// POUs/BACnet Objects/Local (Server)/ADS/FB_BACnet_BinaryOutput_ADS
FUNCTION_BLOCK FB_BACnet_BinaryOutput_ADS
VAR_INPUT
	bEnablePV			: BOOL; (* enable PV write commands *)
	bNullPV				: BOOL; (* clear priority entry *)
	bPV					: BOOL; (* present value bool type *)
	bManual				: BOOL; (* FALSE --> TRUE: write present_value immediately, FALSE: only write present_value on-change, TRUE: write present_value on-change and when device turns operational *)
	ePriority			: E_BACNETPRIORITY := BACNETPRIORITY_12;
END_VAR
VAR_IN_OUT
	Device				: FB_BACnet_Device;
END_VAR
VAR_OUTPUT
	bReady				: BOOL;
	bPvDone				: BOOL; (* present_value written over ADS *)
	bPresentValue		: BOOL;
	bOverridden			: BOOL;
	bOutOfService		: BOOL;
	bFault				: BOOL;
	bInAlarm			: BOOL;
	tObjectID			: T_BACnet_ObjectIdentifier := 16#FFFFFFFF;
	bError				: BOOL;
	nErrorId			: UINT;
	nAdsErrorId			: UDINT;
END_VAR
VAR
	_ObjectId AT%I*: DWORD;				(* ~(BACnet_ObjectIdentifier	:		: LINK) *)
	_PresentValue AT%I*: WORD; 			(* ~(BACnet_PresentValue 		:		: )
								   			(BACnet_ObjectType 			: BO	: )	*)
    _PresentValue_Ads : WORD;
	_StatusFlags AT%I*: WORD; 			(* ~(BACnet_StatusFlags 		:		: )	*)
	_StatusFlagsBits : ST_BACnet_StatusFlags;
	_nUpdateCount : UDINT := 0;
	_WriteProp : FB_BACnet_WriteProp;
	_rtrigManual : R_TRIG;
	_bNullPvOld : BOOL;
	_nObjType : E_BACNETOBJECTTYPE;
END_VAR

(* update server device *)
IF (Device._nUpdateCount = _nUpdateCount) THEN
	Device();
END_IF
(* remind current number of update counter *)
_nUpdateCount := Device._nUpdateCount;

(* trigger on manual flag *)
_rtrigManual(CLK:= bManual, Q=> );

(* decode object type *)
_nObjType := F_BACnet_GetObjType(_ObjectId);

IF Device.bFirstCycle THEN
	(* first call of the server device since reboot/reset *)
	bReady := FALSE;
	bPvDone := FALSE;

ELSIF _nObjType <> BACnetObjectType_BinaryOutput THEN
	(* wrong mapped object type *)
	nErrorId := BACnet_ERR_INVALID_OBJECTTYPE;
	bReady := FALSE;
	bPvDone := FALSE;

ELSIF (_StatusFlags < 4) THEN
	(* wrong mapping *)
	nErrorId := BACnet_ERR_WRONG_MAPPING;
	bReady := FALSE;
	bPvDone := FALSE;

ELSIF Device.bOperational THEN

	IF Device.stAdsConn.bValid THEN
		(* write present_value on manual trigger, on-change and on operational recover *)
		IF	(		bEnablePV
				AND	(		(bPV <> F_BinPV_To_Bool(TO_INT(_PresentValue_Ads)))
						OR	((NOT bReady) AND bManual)
						OR	(bNullPV <> _bNullPvOld)
						OR	_rtrigManual.Q
					)
			)
		THEN
			_WriteProp.bExecute := TRUE;
			bPvDone := FALSE;
			(* write depending on enable state *)
			_PresentValue_Ads := TO_WORD(F_Bool_To_BinPV(TRUE, bNullPV, bPV));
			_bNullPvOld := bNullPV;
		END_IF

		(* ready state *)
		IF (nAdsErrorId = 0) THEN
			bReady := TRUE;
			nErrorId := BACnet_ERR_NO_ERROR;
		END_IF

	ELSE
		(* invalid ADS connection *)
		bReady := FALSE;
		nErrorId := BACnet_ERR_INVALID_ADS_CONN;
		bPvDone := FALSE;
	END_IF


	(* present value *)
	bPresentValue := F_BinPV_To_Bool(TO_INT(_PresentValue));

	(* build bit states *)
	_StatusFlagsBits := F_BACnet_StatusFlags(_StatusFlags);

	(* copy states to output *)
	bOverridden := _StatusFlagsBits.overridden;
	bOutOfService := _StatusFlagsBits.out_of_service;
	bFault := _StatusFlagsBits.fault;
	bInAlarm := _StatusFlagsBits.in_alarm;
	tObjectID := _ObjectId;

ELSE
	(* server device not ready, reset local ready also *)
	bReady := FALSE;
	nErrorId := BACnet_ERR_OPERATIONAL;
	bPvDone := FALSE;
END_IF

(* call write property command *)
_WriteProp(
	BACnetDevicePort	:= Device.stAdsConn.nAmsPort,
	bExecute			:= ,
	sNetId				:= Device.stAdsConn.sAmsNetId,
	ObjectType			:= _nObjType,
	PropertyID			:= BACnetPropertyIdentifier_PresentValue,
	Priority			:= ePriority,
	DataType			:= BACnetDataType_BinaryPV,
	ObjectInstance		:= F_BACnet_GetObjInstance(_ObjectId),
	ptrValue			:= ADR(_PresentValue_Ads),
	nLenValue			:= SIZEOF(_PresentValue_Ads),
	bDone				=> ,
	bBusy				=> ,
	bError				=> ,
	nErrID				=> );

(* set done flag *)
IF _WriteProp.bExecute AND (NOT _WriteProp.bBusy) THEN
	(* check if command was finished with error *)
	IF _WriteProp.bError THEN
		bPvDone		:= FALSE;
		bReady		:= FALSE;
		nErrorId	:= BACnet_ERR_ADS_Write;
	ELSE
		(* successful written *)
		bPvDone		:= TRUE;
	END_IF
	nAdsErrorId := _WriteProp.nErrID;
	(* reset execution bit *)
	_WriteProp(bExecute := FALSE);
END_IF

(* set error flag *)
bError := (nErrorId <> BACnet_ERR_NO_ERROR) OR (nAdsErrorId <> 0);

END_FUNCTION_BLOCK

// POUs/BACnet Objects/Local (Server)/ADS/FB_BACnet_BinaryValue_ADS
FUNCTION_BLOCK FB_BACnet_BinaryValue_ADS
VAR_INPUT
	bEnablePV			: BOOL; (* enable PV write commands *)
	bNullPV				: BOOL; (* clear priority entry *)
	bPV					: BOOL; (* present value bool type *)
	bManual				: BOOL; (* FALSE --> TRUE: write present_value immediately, FALSE: only write present_value on-change, TRUE: write present_value on-change and when device turns operational *)
	ePriority			: E_BACNETPRIORITY := BACNETPRIORITY_12;
END_VAR
VAR_IN_OUT
	Device				: FB_BACnet_Device;
END_VAR
VAR_OUTPUT
	bReady				: BOOL;
	bPvDone				: BOOL; (* present_value written over ADS *)
	bPresentValue		: BOOL;
	bOverridden			: BOOL;
	bOutOfService		: BOOL;
	bFault				: BOOL;
	bInAlarm			: BOOL;
	tObjectID			: T_BACnet_ObjectIdentifier := 16#FFFFFFFF;
	bError				: BOOL;
	nErrorId			: UINT;
	nAdsErrorId			: UDINT;
END_VAR
VAR
	_ObjectId AT%I*: DWORD;				(* ~(BACnet_ObjectIdentifier		:		: LINK) *)
	_PresentValue AT%I*: WORD; 			(* ~(BACnet_PresentValue 			:		: )
								   			(BACnet_ObjectType 				: BV	: )	*)
    _PresentValue_Ads : WORD;
	_StatusFlags AT%I*: WORD; 			(* ~(BACnet_StatusFlags 			:		: )	*)
	_StatusFlagsBits : ST_BACnet_StatusFlags;
	_nUpdateCount : UDINT := 0;
	_WriteProp : FB_BACnet_WriteProp;
	_rtrigManual : R_TRIG;
	_bNullPvOld : BOOL;
	_nObjType : E_BACNETOBJECTTYPE;
END_VAR

(* update server device *)
IF (Device._nUpdateCount = _nUpdateCount) THEN
	Device();
END_IF
(* remind current number of update counter *)
_nUpdateCount := Device._nUpdateCount;

(* trigger on manual flag *)
_rtrigManual(CLK:= bManual, Q=> );

(* decode object type *)
_nObjType := F_BACnet_GetObjType(_ObjectId);

IF Device.bFirstCycle THEN
	(* first call of the server device since reboot/reset *)
	bReady := FALSE;
	bPvDone := FALSE;

ELSIF _nObjType <> BACnetObjectType_BinaryValue THEN
	(* wrong mapped object type *)
	nErrorId := BACnet_ERR_INVALID_OBJECTTYPE;
	bReady := FALSE;
	bPvDone := FALSE;

ELSIF (_StatusFlags < 4) THEN
	(* wrong mapping *)
	nErrorId := BACnet_ERR_WRONG_MAPPING;
	bReady := FALSE;
	bPvDone := FALSE;

ELSIF Device.bOperational THEN

	IF Device.stAdsConn.bValid THEN
		(* write present_value on manual trigger, on-change and on operational recover *)
		IF (		bEnablePV
				AND	(		(bPV <> F_BinPV_To_Bool(TO_INT(_PresentValue_Ads)))
						OR	((NOT bReady) AND bManual)
						OR	(bNullPV <> _bNullPvOld)
						OR	_rtrigManual.Q
					)
			)
		THEN
			_WriteProp.bExecute := TRUE;
			bPvDone := FALSE;
			(* write depending on enable state *)
			_PresentValue_Ads := to_word(F_Bool_To_BinPV(TRUE, bNullPV, bPV));
			_bNullPvOld := bNullPV;
		END_IF

		(* ready state *)
		IF (nAdsErrorId = 0) THEN
			bReady := TRUE;
			nErrorId := BACnet_ERR_NO_ERROR;
		END_IF

	ELSE
		(* invalid ADS connection *)
		bReady := FALSE;
		nErrorId := BACnet_ERR_INVALID_ADS_CONN;
		bPvDone := FALSE;
	END_IF

	(* present value *)
	bPresentValue := F_BinPV_To_Bool(TO_INT(_PresentValue));

	(* build bit states *)
	_StatusFlagsBits := F_BACnet_StatusFlags(_StatusFlags);

	(* copy states to output *)
	bOverridden := _StatusFlagsBits.overridden;
	bOutOfService := _StatusFlagsBits.out_of_service;
	bFault := _StatusFlagsBits.fault;
	bInAlarm := _StatusFlagsBits.in_alarm;
	tObjectID := _ObjectId;

ELSE
	(* server device not ready, reset local ready also *)
	bReady := FALSE;
	nErrorId := BACnet_ERR_OPERATIONAL;
	bPvDone := FALSE;
END_IF

(* call write property command *)
_WriteProp(
	BACnetDevicePort	:= Device.stAdsConn.nAmsPort,
	bExecute			:= ,
	sNetId				:= Device.stAdsConn.sAmsNetId,
	ObjectType			:= _nObjType,
	PropertyID			:= BACnetPropertyIdentifier_PresentValue,
	Priority			:= ePriority,
	DataType			:= BACnetDataType_BinaryPV,
	ObjectInstance		:= F_BACnet_GetObjInstance(_ObjectId),
	ptrValue			:= ADR(_PresentValue_Ads),
	nLenValue			:= SIZEOF(_PresentValue_Ads),
	bDone				=> ,
	bBusy				=> ,
	bError				=> ,
	nErrID				=> );

(* set done flag *)
IF _WriteProp.bExecute AND (NOT _WriteProp.bBusy) THEN
	(* check if command was finished with error *)
	IF _WriteProp.bError THEN
		bPvDone		:= FALSE;
		bReady		:= FALSE;
		nErrorId	:= BACnet_ERR_ADS_Write;
	ELSE
		(* successful written *)
		bPvDone		:= TRUE;
	END_IF
	nAdsErrorId := _WriteProp.nErrID;
	(* reset execution bit *)
	_WriteProp(bExecute := FALSE);
END_IF

(* set error flag *)
bError := (nErrorId <> BACnet_ERR_NO_ERROR) OR (nAdsErrorId <> 0);

END_FUNCTION_BLOCK

// POUs/BACnet Objects/Local (Server)/ADS/FB_BACnet_MultiStateOutput_ADS
FUNCTION_BLOCK FB_BACnet_MultiStateOutput_ADS
VAR_INPUT
	bEnablePV			: BOOL; (* enable PV write commands *)
	bNullPV				: BOOL; (* clear priority entry *)
	nPV					: UDINT; (* number for priority x, when input bEnablePV is TRUE and bNullPV is FALSE *)
	bManual				: BOOL; (* FALSE --> TRUE: write present_value immediately, FALSE: only write present_value on-change, TRUE: write present_value on-change and when device turns operational *)
	ePriority			: E_BACNETPRIORITY := BACNETPRIORITY_12;
END_VAR
VAR_IN_OUT
	Device				: FB_BACnet_Device;
END_VAR
VAR_OUTPUT
	bReady				: BOOL;
	bPvDone				: BOOL; (* present_value written over ADS *)
	nPresentValue		: UDINT;
	bOverridden			: BOOL;
	bOutOfService		: BOOL;
	bFault				: BOOL;
	bInAlarm			: BOOL;
	nNbrOfStates		: UDINT;
	tObjectID			: T_BACnet_ObjectIdentifier := 16#FFFFFFFF;
	bError				: BOOL;
	nErrorId			: UINT;
	nAdsErrorId			: UDINT;
END_VAR
VAR
	_StatusFlags AT%I*: WORD; 				(* ~(BACnet_StatusFlags			:		: )	*)
	_PresentValue AT%I*: UDINT; 			(* ~(BACnet_PresentValue 		:		: )
								   				(BACnet_ObjectType			: MO	: )	*)
	_NumberOfStates AT%I*: UDINT;			(* ~(BACnet_NumberOfStates		:		: )	*)
	_ObjectId AT%I*: DWORD;					(* ~(BACnet_ObjectIdentifier	:		: LINK) *)
	_StatusFlagsBits : ST_BACnet_StatusFlags;
    _PresentValue_Ads : UDINT;
	_nUpdateCount : UDINT := 0;
	_WriteProp : FB_BACnet_WriteProp;
	_rtrigManual : R_TRIG;
	_bNullPvOld : BOOL;
	_nObjType : E_BACNETOBJECTTYPE;
END_VAR

(* update server device *)
IF (Device._nUpdateCount = _nUpdateCount) THEN
	Device();
END_IF
(* remind current number of update counter *)
_nUpdateCount := Device._nUpdateCount;

(* trigger on manual flag *)
_rtrigManual(CLK:= bManual, Q=> );

(* decode object type *)
_nObjType := F_BACnet_GetObjType(_ObjectId);

IF Device.bFirstCycle THEN
	(* first call of the server device since reboot/reset *)
	bReady := FALSE;
	bPvDone := FALSE;

ELSIF _nObjType <> BACnetObjectType_MultiStateOutput THEN
	(* wrong mapped object type *)
	nErrorId := BACnet_ERR_INVALID_OBJECTTYPE;
	bReady := FALSE;
	bPvDone := FALSE;

ELSIF (_StatusFlags < 4) THEN
	(* wrong mapping *)
	nErrorId := BACnet_ERR_WRONG_MAPPING;
	bReady := FALSE;
	bPvDone := FALSE;

ELSIF Device.bOperational THEN

	IF Device.stAdsConn.bValid THEN
		(* write present_value on manual trigger, on-change and on operational recover *)
		IF		bEnablePV
			AND	(		_rtrigManual.Q
					OR	(nPV <> _PresentValue_Ads)
					OR	((NOT bReady) AND bManual)
					OR	(bNullPV <> _bNullPvOld)
				)
		THEN
			_WriteProp.bExecute := TRUE;
			bPvDone := FALSE;
			(* write depending on enable state *)
			IF bNullPV THEN
				_PresentValue_Ads := 0;
			ELSE
				_PresentValue_Ads := nPV;
			END_IF
			_bNullPvOld := bNullPV;
		END_IF

		(* ready state *)
		IF (nAdsErrorId = 0) THEN
			bReady := TRUE;
			nErrorId := BACnet_ERR_NO_ERROR;
		END_IF

	ELSE
		(* invalid ADS connection *)
		bReady := FALSE;
		nErrorId := BACnet_ERR_INVALID_ADS_CONN;
		bPvDone := FALSE;
	END_IF

	(* present value *)
	nPresentValue := _PresentValue;

	(* build bit states *)
	_StatusFlagsBits := F_BACnet_StatusFlags(_StatusFlags);

	(* copy states to output *)
	bOverridden := _StatusFlagsBits.overridden;
	bOutOfService := _StatusFlagsBits.out_of_service;
	bFault := _StatusFlagsBits.fault;
	bInAlarm := _StatusFlagsBits.in_alarm;
	tObjectID := _ObjectId;

	(* number of states *)
	nNbrOfStates := _NumberOfStates;

ELSE
	(* server device not ready, reset local ready also *)
	bReady := FALSE;
	nErrorId := BACnet_ERR_OPERATIONAL;
	bPvDone := FALSE;
END_IF

(* call write property command *)
_WriteProp(
	BACnetDevicePort	:= Device.stAdsConn.nAmsPort,
	bExecute			:= ,
	sNetId				:= Device.stAdsConn.sAmsNetId,
	ObjectType			:= _nObjType,
	PropertyID			:= BACnetPropertyIdentifier_PresentValue,
	Priority			:= ePriority,
	DataType			:= BACnetDataType_UnsignedInteger,
	ObjectInstance		:= F_BACnet_GetObjInstance(_ObjectId),
	ptrValue			:= ADR(_PresentValue_Ads),
	nLenValue			:= SIZEOF(_PresentValue_Ads),
	bDone				=> ,
	bBusy				=> ,
	bError				=> ,
	nErrID				=> );

(* set done flag *)
IF _WriteProp.bExecute AND (NOT _WriteProp.bBusy) THEN
	(* check if command was finished with error *)
	IF _WriteProp.bError THEN
		bPvDone		:= FALSE;
		bReady		:= FALSE;
		nErrorId	:= BACnet_ERR_ADS_Write;
	ELSE
		(* successful written *)
		bPvDone		:= TRUE;
	END_IF
	nAdsErrorId := _WriteProp.nErrID;
	(* reset execution bit *)
	_WriteProp(bExecute := FALSE);
END_IF

(* set error flag *)
bError := (nErrorId <> BACnet_ERR_NO_ERROR) OR (nAdsErrorId <> 0);

END_FUNCTION_BLOCK

// POUs/BACnet Objects/Local (Server)/ADS/FB_BACnet_MultiStateValue_ADS
FUNCTION_BLOCK FB_BACnet_MultiStateValue_ADS
VAR_INPUT
	bEnablePV			: BOOL; (* enable PV write commands *)
	bNullPV				: BOOL; (* clear priority entry *)
	nPV					: UDINT; (* number for priority x, when input bEnablePV is TRUE and bNullPV is FALSE *)
	bManual				: BOOL; (* FALSE --> TRUE: write present_value immediately, FALSE: only write present_value on-change, TRUE: write present_value on-change and when device turns operational *)
	ePriority			: E_BACNETPRIORITY := BACNETPRIORITY_12;
END_VAR
VAR_IN_OUT
	Device				: FB_BACnet_Device;
END_VAR
VAR_OUTPUT
	bReady				: BOOL;
	bPvDone				: BOOL; (* present_value written over ADS *)
	nPresentValue		: UDINT;
	bOverridden			: BOOL;
	bOutOfService		: BOOL;
	bFault				: BOOL;
	bInAlarm			: BOOL;
	nNbrOfStates		: UDINT;
	tObjectID			: T_BACnet_ObjectIdentifier := 16#FFFFFFFF;
	bError				: BOOL;
	nErrorId			: UINT;
	nAdsErrorId			: UDINT;
END_VAR
VAR
	_StatusFlags AT%I*: WORD; 				(* ~(BACnet_StatusFlags 	:		: )	*)
	_PresentValue AT%I*: UDINT; 			(* ~(BACnet_PresentValue 	:		: )
								   				(BACnet_ObjectType 		: MV	: )	*)
	_NumberOfStates AT%I*: UDINT;			(* ~(BACnet_NumberOfStates	:		: )	*)
	_ObjectId AT%I*: DWORD;					(* ~(BACnet_ObjectIdentifier:		: LINK) *)
	_StatusFlagsBits : ST_BACnet_StatusFlags;
    _PresentValue_Ads : UDINT;
	_nUpdateCount : UDINT := 0;
	_WriteProp : FB_BACnet_WriteProp;
	_rtrigManual : R_TRIG;
	_bNullPvOld : BOOL;
	_nObjType : E_BACNETOBJECTTYPE;
END_VAR

(* update server device *)
IF (Device._nUpdateCount = _nUpdateCount) THEN
	Device();
END_IF
(* remind current number of update counter *)
_nUpdateCount := Device._nUpdateCount;

(* trigger on manual flag *)
_rtrigManual(CLK:= bManual, Q=> );

(* decode object type *)
_nObjType := F_BACnet_GetObjType(_ObjectId);

IF Device.bFirstCycle THEN
	(* first call of the server device since reboot/reset *)
	bReady := FALSE;
	bPvDone := FALSE;

ELSIF _nObjType <> BACnetObjectType_MultiStateValue THEN
	(* wrong mapped object type *)
	nErrorId := BACnet_ERR_INVALID_OBJECTTYPE;
	bReady := FALSE;
	bPvDone := FALSE;

ELSIF (_StatusFlags < 4) THEN
	(* wrong mapping *)
	nErrorId := BACnet_ERR_WRONG_MAPPING;
	bReady := FALSE;
	bPvDone := FALSE;

ELSIF Device.bOperational THEN

	IF Device.stAdsConn.bValid THEN
		(* write present_value on manual trigger, on-change and on operational recover *)
		IF		bEnablePV
			AND	(		_rtrigManual.Q
					OR	(nPV <> _PresentValue_Ads)
					OR	((NOT bReady) AND bManual)
					OR	(bNullPV <> _bNullPvOld)
				)
		THEN
			_WriteProp.bExecute := TRUE;
			bPvDone := FALSE;
			(* write depending on enable state *)
			IF bNullPV THEN
				_PresentValue_Ads := 0;
			ELSE
				_PresentValue_Ads := nPV;
			END_IF
			_bNullPvOld := bNullPV;
		END_IF

		(* ready state *)
		IF (nAdsErrorId = 0) THEN
			bReady := TRUE;
			nErrorId := BACnet_ERR_NO_ERROR;
		END_IF

	ELSE
		(* invalid ADS connection *)
		bReady := FALSE;
		nErrorId := BACnet_ERR_INVALID_ADS_CONN;
		bPvDone := FALSE;
	END_IF

	(* present value *)
	nPresentValue := _PresentValue;

	(* build bit states *)
	_StatusFlagsBits := F_BACnet_StatusFlags(_StatusFlags);

	(* copy states to output *)
	bOverridden := _StatusFlagsBits.overridden;
	bOutOfService := _StatusFlagsBits.out_of_service;
	bFault := _StatusFlagsBits.fault;
	bInAlarm := _StatusFlagsBits.in_alarm;
	tObjectID := _ObjectId;

	(* number of states *)
	nNbrOfStates := _NumberOfStates;

ELSE
	(* server device not ready, reset local ready also *)
	bReady := FALSE;
	nErrorId := BACnet_ERR_OPERATIONAL;
	bPvDone := FALSE;
END_IF

(* call write property command *)
_WriteProp(
	BACnetDevicePort	:= Device.stAdsConn.nAmsPort,
	bExecute			:= ,
	sNetId				:= Device.stAdsConn.sAmsNetId,
	ObjectType			:= _nObjType,
	PropertyID			:= BACnetPropertyIdentifier_PresentValue,
	Priority			:= ePriority,
	DataType			:= BACnetDataType_UnsignedInteger,
	ObjectInstance		:= F_BACnet_GetObjInstance(_ObjectId),
	ptrValue			:= ADR(_PresentValue_Ads),
	nLenValue			:= SIZEOF(_PresentValue_Ads),
	bDone				=> ,
	bBusy				=> ,
	bError				=> ,
	nErrID				=> );

(* set done flag *)
IF _WriteProp.bExecute AND (NOT _WriteProp.bBusy) THEN
	(* check if command was finished with error *)
	IF _WriteProp.bError THEN
		bPvDone		:= FALSE;
		bReady		:= FALSE;
		nErrorId	:= BACnet_ERR_ADS_Write;
	ELSE
		(* successful written *)
		bPvDone		:= TRUE;
	END_IF
	nAdsErrorId := _WriteProp.nErrID;
	(* reset execution bit *)
	_WriteProp(bExecute := FALSE);
END_IF

(* set error flag *)
bError := (nErrorId <> BACnet_ERR_NO_ERROR) OR (nAdsErrorId <> 0);

END_FUNCTION_BLOCK

// POUs/BACnet Objects/Local (Server)/DRV/FB_BACnet_Loop_DRV
FUNCTION_BLOCK FB_BACnet_Loop_DRV
VAR_IN_OUT
	Device	: FB_BACnet_Device;
END_VAR
VAR_OUTPUT
	bReady				: BOOL;
	fSetPoint			: REAL;
	fControlledValue	: REAL;
	fPresentValue		: REAL;
	bOverridden			: BOOL;
	bOutOfService		: BOOL;
	bFault				: BOOL;
	bInAlarm			: BOOL;
	bError				: BOOL;
	nErrorId			: UINT;
END_VAR
VAR
	_ControlledVariableValue AT%I*: REAL;	(* ~(BACnet_ControlledVariableValue :		: )
												(BACnet_ObjectType				: LOOP	: )
												(BACnet_EnableInternalLoopCtrl	: TRUE	: NOLINK,ENABLE) *)
	_Setpoint AT%I*:REAL;					(* ~(BACnet_Setpoint				:		: )	*)
	_PresentValue AT%I*: REAL; 				(* ~(BACnet_PresentValue 			: 		: )	*)
	_ObjectId AT%I*: DWORD;					(* ~(BACnet_ObjectIdentifier		:		: LINK) *)
	_StatusFlags AT%I*: WORD; 				(* ~(BACnet_StatusFlags 			: 		: )	*)
	_StatusFlagsBits : ST_BACnet_StatusFlags;
	_nUpdateCount : UDINT := 0;
END_VAR

(* update server device *)
IF (Device._nUpdateCount = _nUpdateCount) THEN
	Device();
END_IF
(* remind current number of update counter *)
_nUpdateCount := Device._nUpdateCount;

(* check BitString format of StatusFlags --> if StatusFlags are less than 4, object isn't linked correctly *)
IF (_StatusFlags < 4) THEN
	(* wrong mapping *)
	nErrorId := BACnet_ERR_WRONG_MAPPING;
	bReady := FALSE;

ELSIF Device.bOperational THEN
	(* ready state *)
	bReady := TRUE;
	nErrorId := BACnet_ERR_NO_ERROR;

	(* decode status flags *)
	_StatusFlagsBits := F_BACnet_StatusFlags(_StatusFlags);

	(* copy states to output *)
	bOverridden := _StatusFlagsBits.overridden;
	bOutOfService := _StatusFlagsBits.out_of_service;
	bFault := _StatusFlagsBits.fault;
	bInAlarm := _StatusFlagsBits.in_alarm;

	(* set other outputs *)
	fSetPoint := _Setpoint;
	fPresentValue := _PresentValue;
	fControlledValue := _ControlledVariableValue;
ELSE
	(* server device not ready, reset local ready also *)
	bReady := FALSE;
	nErrorId := BACnet_ERR_OPERATIONAL;
END_IF
(* set error flag *)
bError := (nErrorId <> BACnet_ERR_NO_ERROR);

END_FUNCTION_BLOCK

// POUs/BACnet Objects/Local (Server)/DRV/FB_BACnet_Loop_DRV_EX
FUNCTION_BLOCK FB_BACnet_Loop_DRV_EX
VAR_IN_OUT
	Device	: FB_BACnet_Device;
END_VAR
VAR_OUTPUT
	bReady				: BOOL;
	fSetPoint			: REAL;
	fControlledValue	: REAL;
	fPresentValue		: REAL;
	fPropBand			: REAL; (* controller output in range of -100...100% in relation to Min.-/Max.-output *)
	bOverridden			: BOOL;
	bOutOfService		: BOOL;
	bFault				: BOOL;
	bInAlarm			: BOOL;
	bOpenLoop			: BOOL;
	bCommFailure		: BOOL;
	bOtherFault			: BOOL;
	eEventState			: E_BACNETEVENTSTATE;
	bAckedTrans_ToOffNormal : BOOL;
	bAckedTrans_ToFault		: BOOL;
	bAckedTrans_ToNormal	: BOOL;
	tObjectID			: T_BACnet_ObjectIdentifier := 16#FFFFFFFF;
	bError				: BOOL;
	nErrorId			: UINT;
END_VAR
VAR
	_ControlledVariableValue AT%I*: REAL;	(* ~(BACnet_ControlledVariableValue :		: )
												(BACnet_ObjectType				: LOOP	: )
												(BACnet_EnableInternalLoopCtrl	: TRUE	: NOLINK,ENABLE) *)
	_Setpoint AT%I*:REAL;					(* ~(BACnet_Setpoint				:		: )	*)
	_MaximumOutput AT%I*:REAL;				(* ~(BACnet_MaximumOutput			:		: )	*)
	_MinimumOutput AT%I*:REAL;				(* ~(BACnet_MinimumOutput			:		: )	*)
	_PresentValue AT%I*: REAL; 				(* ~(BACnet_PresentValue 			: 		: )	*)
	_ObjectId AT%I*: DWORD;					(* ~(BACnet_ObjectIdentifier		:		: LINK) *)
	_StatusFlags AT%I*: WORD; 				(* ~(BACnet_StatusFlags 			: 		: )	*)
	_AckedTransitions AT%I*:WORD;			(* ~(BACnet_AckedTransitions		:		: ) *)
	_EventState AT%I*: WORD; 				(* ~(BACnet_EventState 				:		: )	*)
	_Reliability AT%I*: WORD;(* ~(BACNET_RELIABILITY 			:		: )	*)
	_StatusFlagsBits : ST_BACnet_StatusFlags;
	_AckedTransBits : ST_BACnet_EventTransitionBits;
	_nUpdateCount : UDINT := 0;
END_VAR

(* update server device *)
IF (Device._nUpdateCount = _nUpdateCount) THEN
	Device();
END_IF
(* remind current number of update counter *)
_nUpdateCount := Device._nUpdateCount;

(* check BitString format of StatusFlags --> if StatusFlags are less than 4, object isn't linked correctly *)
IF (F_BACnet_GetObjType(_ObjectId) <> BACnetObjectType_Loop) THEN
	(* wrong mapping / invalid object ID *)
	IF _ObjectId = 0 THEN
		nErrorId := BACnet_ERR_WRONG_MAPPING;
	ELSE
		nErrorId := BACnet_ERR_INVALID_OBJECTID;
	END_IF
	bReady := FALSE;
	tObjectID := 16#FFFFFFFF;

ELSIF (_StatusFlags < 4) THEN
	(* wrong mapping *)
	nErrorId := BACnet_ERR_WRONG_MAPPING;
	bReady := FALSE;

ELSIF Device.bOperational THEN
	(* ready state *)
	bReady := TRUE;
	nErrorId := BACnet_ERR_NO_ERROR;

	(* decode status flags *)
	_StatusFlagsBits := F_BACnet_StatusFlags(_StatusFlags);
	_AckedTransBits	:= F_BACnet_EventTransitionFlags(_AckedTransitions);

	(* copy states to output *)
	bOverridden := _StatusFlagsBits.overridden;
	bOutOfService := _StatusFlagsBits.out_of_service;
	bFault := _StatusFlagsBits.fault;
	bInAlarm := _StatusFlagsBits.in_alarm;
	bOpenLoop := _Reliability = TO_WORD(BACnetReliability_open_loop);
	bCommFailure := _Reliability = TO_WORD(BACnetReliability_communication_failure);
	bOtherFault := _Reliability = TO_WORD(BACnetReliability_unreliable_other);
	bAckedTrans_ToOffNormal := _AckedTransBits.to_offnormal;
	bAckedTrans_ToFault := _AckedTransBits.to_fault;
	bAckedTrans_ToNormal := _AckedTransBits.to_normal;
	tObjectID := _ObjectId;
	eEventState := TO_INT(_EventState);

	(* calculate proportional band *)
	IF (_MaximumOutput > 0.0) AND (_MinimumOutput >= 0.0) THEN
		fPropBand := ((_PresentValue - _MinimumOutput) / (_MaximumOutput - _MinimumOutput)) * 100.0;
	ELSIF (_MaximumOutput <= 0.0) AND (_MinimumOutput < 0.0) THEN
		fPropBand := ((_PresentValue - _MaximumOutput) / (_MaximumOutput - _MinimumOutput)) * 100.0;
	ELSIF (_PresentValue > 0.0) AND (_MaximumOutput > 0.0) THEN
		fPropBand := (_PresentValue / _MaximumOutput) * 100.0;
	ELSIF (_PresentValue < 0.0) AND (_MinimumOutput < 0.0) THEN
		fPropBand := (_PresentValue / _MinimumOutput) * -100.0;
	ELSE
		fPropBand := 0.0;
	END_IF

	(* set other outputs *)
	fSetPoint := _Setpoint;
	fPresentValue := _PresentValue;
	fControlledValue := _ControlledVariableValue;
ELSE
	(* server device not ready, reset local ready also *)
	bReady := FALSE;
	nErrorId := BACnet_ERR_OPERATIONAL;
END_IF
(* set error flag *)
bError := (nErrorId <> BACnet_ERR_NO_ERROR);

END_FUNCTION_BLOCK

// POUs/BACnet Objects/Local (Server)/Extended Process Data/FB_BACnet_Accumulator_EX
FUNCTION_BLOCK FB_BACnet_Accumulator_EX
VAR_INPUT
	nPV					: UDINT; (* number for present_value *)
END_VAR
VAR_IN_OUT
	Device				: FB_BACnet_Device;
END_VAR
VAR_OUTPUT
	bReady				: BOOL;
	nPresentValue		: UDINT;
	nMaxPV				: UDINT;
	bOverridden			: BOOL;
	bOutOfService		: BOOL;
	bFault				: BOOL;
	bInAlarm			: BOOL;
	bOverRange			: BOOL;
	bUnderRange			: BOOL;
	bNoSensor			: BOOL;
	bOpenLoop			: BOOL;
	bCommFailure		: BOOL;
	bShortedLoop		: BOOL;
	bOtherFault			: BOOL;
	eEventState			: E_BACNETEVENTSTATE;
	tObjectID			: T_BACnet_ObjectIdentifier := 16#FFFFFFFF;
	bError				: BOOL;
	nErrorId			: UINT;
END_VAR
VAR
	_PresentValueIn AT%I*:UDINT;	(* ~(BACnet_PresentValue	:		: )
										(BACnet_ObjectType		: ACC	: )	*)
    _PresentValueOut AT%Q*:UDINT;	(* ~(BACnet_PresentValue	:		: )	*)
	_MaxPresValue AT%I*:UDINT;		(* ~(BACnet_MaxPresValue	:		: writeprotect) *)
	_ObjectId AT%I*: DWORD;			(* ~(BACnet_ObjectIdentifier:		: LINK) *)
	_StatusFlags AT%I*:WORD;		(* ~(BACnet_StatusFlags		:		: )	*)
	_EventState AT%I*: WORD; 		(* ~(BACnet_EventState 		:		: )	*)
	_Reliability AT%I*: WORD;; 		(* ~(BACnet_Reliability 	:		: )	*)
	_nUpdateCount : UDINT := 0;
	_StatusFlagsBits : ST_BACnet_StatusFlags;
END_VAR

(* update client device *)
IF (Device._nUpdateCount = _nUpdateCount) THEN
	Device();
END_IF
(* remind current number of update counter *)
_nUpdateCount := Device._nUpdateCount;

(* check object type *)
IF (F_BACnet_GetObjType(_ObjectId) <> BACnetObjectType_Accumulator) THEN
	(* wrong mapping / invalid object ID *)
	IF _ObjectId = 0 THEN
		nErrorId := BACnet_ERR_WRONG_MAPPING;
	ELSE
		nErrorId := BACnet_ERR_INVALID_OBJECTID;
	END_IF
	bReady := FALSE;

ELSIF _StatusFlags < 4 THEN
	(* mapping seems to be wrong (bit string for status flags must be 4 in minimum) *)
	nErrorId := BACnet_ERR_WRONG_MAPPING;

ELSIF Device.bOperational THEN
	(* clear error flag *)
	nErrorId := BACnet_ERR_NO_ERROR;
	bReady := TRUE;
	(* copy present value *)
	nPresentValue 		:= _PresentValueIn;
	_PresentValueOut	:= nPV;
	nMaxPV				:= _MaxPresValue;

	(* build bit states *)
	_StatusFlagsBits	:= F_BACnet_StatusFlags(_StatusFlags);

	(* copy states to output *)
	bOverridden := _StatusFlagsBits.overridden;
	bOutOfService := _StatusFlagsBits.out_of_service;
	bFault := _StatusFlagsBits.fault;
	bInAlarm := _StatusFlagsBits.in_alarm;
	bOverRange := (_Reliability = TO_WORD(BACnetReliability_over_range));
	bUnderRange := (_Reliability = TO_WORD(BACnetReliability_under_range));
	bNoSensor := (_Reliability = TO_WORD(BACnetReliability_no_sensor));
	bOpenLoop := (_Reliability = TO_WORD(BACnetReliability_open_loop));
	bCommFailure := (_Reliability = TO_WORD(BACnetReliability_communication_failure));
	bShortedLoop := (_Reliability = TO_WORD(BACnetReliability_shorted_loop));
	bOtherFault := (_Reliability = TO_WORD(BACnetReliability_unreliable_other));
	tObjectID := _ObjectId;

	(* convert enumeration *)
	eEventState := TO_INT(_EventState);
ELSE
	bReady := FALSE;
	(* and set error ID *)
	nErrorId := BACnet_ERR_OPERATIONAL;
END_IF

(* set error flag *)
bError := (nErrorId <> BACnet_ERR_NO_ERROR);

END_FUNCTION_BLOCK

// POUs/BACnet Objects/Local (Server)/Extended Process Data/FB_BACnet_AnalogInput_EX
FUNCTION_BLOCK FB_BACnet_AnalogInput_EX
VAR_IN_OUT
	Device				: FB_BACnet_Device;
END_VAR
VAR_OUTPUT
	bReady				: BOOL;
	fPresentValue		: REAL;
	bOverridden			: BOOL;
	bOutOfService		: BOOL;
	bFault				: BOOL;
	bInAlarm			: BOOL;
	bOverRange			: BOOL;
	bUnderRange			: BOOL;
	bNoSensor			: BOOL;
	bOpenLoop			: BOOL;
	bShortedLoop		: BOOL;
	bOtherFault			: BOOL;
	eEventState			: E_BACNETEVENTSTATE;
	bAckedTrans_ToOffNormal : BOOL;
	bAckedTrans_ToFault		: BOOL;
	bAckedTrans_ToNormal	: BOOL;
	tObjectID			: T_BACnet_ObjectIdentifier := 16#FFFFFFFF;
	bError				: BOOL;
	nErrorId			: UINT;
END_VAR
VAR
	_PresentValue AT%I*: REAL; 			(* ~(BACnet_PresentValue 	:		: )
								   			(BACnet_ObjectType 		: AI	: )	*)
	_ObjectId AT%I*: DWORD;				(* ~(BACnet_ObjectIdentifier:		: LINK) *)
	_StatusFlags AT%I*: WORD; 			(* ~(BACnet_StatusFlags 	:		: )	*)
	_EventState AT%I*: WORD; 			(* ~(BACnet_EventState 		:		: )	*)
	_Reliability AT%I*: WORD;; 			(* ~(BACnet_Reliability 	:		: )	*)
	_AckedTransitions AT%I*:WORD;		(* ~(BACnet_AckedTransitions:		: ) *)
	_AckedTransBits : ST_BACnet_EventTransitionBits;
	_StatusFlagsBits : ST_BACnet_StatusFlags;
	_nUpdateCount : UDINT := 0;
END_VAR

(* update server device *)
IF (Device._nUpdateCount = _nUpdateCount) THEN
	Device();
END_IF
(* remind current number of update counter *)
_nUpdateCount := Device._nUpdateCount;

(* check object type *)
IF (F_BACnet_GetObjType(_ObjectId) <> BACnetObjectType_AnalogInput) THEN
	(* wrong mapping / invalid object ID *)
	IF _ObjectId = 0 THEN
		nErrorId := BACnet_ERR_WRONG_MAPPING;
	ELSE
		nErrorId := BACnet_ERR_INVALID_OBJECTID;
	END_IF
	bReady := FALSE;
	tObjectID := 16#FFFFFFFF;

ELSIF (_StatusFlags < 4) THEN
	(* mapping seems to be wrong (bit string for status flags must be 4 in minimum) *)
	(* wrong mapping *)
	nErrorId := BACnet_ERR_WRONG_MAPPING;
	bReady := FALSE;

ELSIF Device.bOperational THEN
	(* ready state *)
	bReady := TRUE;
	nErrorId := BACnet_ERR_NO_ERROR;

	(* present value *)
	fPresentValue := _PresentValue;

	(* build bit states *)
	_StatusFlagsBits := F_BACnet_StatusFlags(_StatusFlags);
	_AckedTransBits		:= F_BACnet_EventTransitionFlags(_AckedTransitions);

	(* copy states to output *)
	bOverridden := _StatusFlagsBits.overridden;
	bOutOfService := _StatusFlagsBits.out_of_service;
	bFault := _StatusFlagsBits.fault;
	bInAlarm := _StatusFlagsBits.in_alarm;
	bOverRange := (_Reliability = TO_WORD(BACnetReliability_over_range));
	bUnderRange := (_Reliability = TO_WORD(BACnetReliability_under_range));
	bNoSensor := (_Reliability = TO_WORD(BACnetReliability_no_sensor));
	bOpenLoop := (_Reliability = TO_WORD(BACnetReliability_open_loop));
	bShortedLoop := (_Reliability = TO_WORD(BACnetReliability_shorted_loop));
	bOtherFault := (_Reliability = TO_WORD(BACnetReliability_unreliable_other));
	bAckedTrans_ToOffNormal := _AckedTransBits.to_offnormal;
	bAckedTrans_ToFault := _AckedTransBits.to_fault;
	bAckedTrans_ToNormal := _AckedTransBits.to_normal;
	tObjectID := _ObjectId;

	(* convert enumeration *)
	eEventState := TO_INT(_EventState);
ELSE
	(* server device not ready, reset local ready also *)
	bReady := FALSE;
	nErrorId := BACnet_ERR_OPERATIONAL;
END_IF
(* set error flag *)
bError := (nErrorId <> BACnet_ERR_NO_ERROR);

END_FUNCTION_BLOCK

// POUs/BACnet Objects/Local (Server)/Extended Process Data/FB_BACnet_AnalogOutput_EX
FUNCTION_BLOCK FB_BACnet_AnalogOutput_EX
VAR_INPUT
	bEnablePV			: BOOL; (* enable present value with priority x in priority array, FALSE = priority x disable *)
	bNullPV				: BOOL; (* clear priority entry *)
	fPV					: REAL; (* decimal number for priority x, when input bEnablePV is TRUE *)
END_VAR
VAR_IN_OUT
	Device				: FB_BACnet_Device;
END_VAR
VAR_OUTPUT
	bReady				: BOOL;
	fPresentValue		: REAL;
	bOverridden			: BOOL;
	bOutOfService		: BOOL;
	bFault				: BOOL;
	bInAlarm			: BOOL;
	bNoOutput			: BOOL;
	bOpenLoop			: BOOL;
	bShortedLoop		: BOOL;
	bOtherFault			: BOOL;
	eEventState			: E_BACNETEVENTSTATE;
	bAckedTrans_ToOffNormal : BOOL;
	bAckedTrans_ToFault		: BOOL;
	bAckedTrans_ToNormal	: BOOL;
	nActivePrio			: UINT;
	tObjectID			: T_BACnet_ObjectIdentifier := 16#FFFFFFFF;
	bError				: BOOL;
	nErrorId			: UINT;
END_VAR
VAR
	_PresentValue AT%I*: REAL; 			(* ~(BACnet_PresentValue 			:		: )
								   			(BACnet_ObjectType 				: AO	: )	*)
    _PresentValue_Priority12 AT%Q*: DWORD;(* ~(BACnet_PresentValue_Priority12:		: )	*)
	_ActivePriority AT%I*: UDINT; 		(* ~(BACnet_ActivePriority 			:		: )	*)
	_ObjectId AT%I*: DWORD;				(* ~(BACnet_ObjectIdentifier		:		: LINK) *)
	_StatusFlags AT%I*: WORD; 			(* ~(BACnet_StatusFlags 			:		: )	*)
	_EventState AT%I*: WORD;			(* ~(BACnet_EventState 				:		: )	*)
	_Reliability AT%I*: WORD;; 			(* ~(BACnet_Reliability 			:		: )	*)
	_AckedTransitions AT%I*:WORD;		(* ~(BACnet_AckedTransitions		:		: ) *)
	_StatusFlagsBits : ST_BACnet_StatusFlags;
	_AckedTransBits : ST_BACnet_EventTransitionBits;
	_nUpdateCount : UDINT := 0;
END_VAR

(* update server device *)
IF (Device._nUpdateCount = _nUpdateCount) THEN
	Device();
END_IF
(* remind current number of update counter *)
_nUpdateCount := Device._nUpdateCount;

IF Device.bFirstCycle THEN
	(* first call of the server device since reboot/reset *)
	bReady := FALSE;
	_PresentValue_Priority12 := F_BACnet_RealNothing();

ELSIF (F_BACnet_GetObjType(_ObjectId) <> BACnetObjectType_AnalogOutput) THEN
	(* wrong mapping / invalid object ID *)
	IF _ObjectId = 0 THEN
		nErrorId := BACnet_ERR_WRONG_MAPPING;
	ELSE
		nErrorId := BACnet_ERR_INVALID_OBJECTID;
	END_IF
	bReady := FALSE;

ELSIF (_StatusFlags < 4) THEN
	(* wrong mapping *)
	nErrorId := BACnet_ERR_WRONG_MAPPING;
	bReady := FALSE;

ELSIF Device.bOperational THEN
	(* ready state *)
	bReady := TRUE;
	nErrorId := BACnet_ERR_NO_ERROR;

	(* write into priority array *)
	_PresentValue_Priority12 := F_BACnet_RealPV(bEnablePV, bNullPV, fPV);

	(* present value *)
	fPresentValue := _PresentValue;

	(* build bit states *)
	_StatusFlagsBits := F_BACnet_StatusFlags(_StatusFlags);
	_AckedTransBits		:= F_BACnet_EventTransitionFlags(_AckedTransitions);

	(* copy states to output *)
	bOverridden := _StatusFlagsBits.overridden;
	bOutOfService := _StatusFlagsBits.out_of_service;
	bFault := _StatusFlagsBits.fault;
	bInAlarm := _StatusFlagsBits.in_alarm;
	bNoOutput := (_Reliability = TO_WORD(BACnetReliability_no_output));
	bOpenLoop := (_Reliability = TO_WORD(BACnetReliability_open_loop));
	bShortedLoop := (_Reliability = TO_WORD(BACnetReliability_shorted_loop));
	bOtherFault := (_Reliability = TO_WORD(BACnetReliability_unreliable_other));
	bAckedTrans_ToOffNormal := _AckedTransBits.to_offnormal;
	bAckedTrans_ToFault := _AckedTransBits.to_fault;
	bAckedTrans_ToNormal := _AckedTransBits.to_normal;
	tObjectID := _ObjectId;

	(* convert enumeration *)
	eEventState := TO_INT(_EventState);

	(* copy active priority *)
	nActivePrio := UDINT_TO_UINT(_ActivePriority);

ELSE
	(* server device not ready, reset local ready also *)
	bReady := FALSE;
	nErrorId := BACnet_ERR_OPERATIONAL;
END_IF
(* set error flag *)
bError := (nErrorId <> BACnet_ERR_NO_ERROR);

END_FUNCTION_BLOCK

// POUs/BACnet Objects/Local (Server)/Extended Process Data/FB_BACnet_AnalogValue_EX
FUNCTION_BLOCK FB_BACnet_AnalogValue_EX
VAR_INPUT
	bEnablePV			: BOOL; (* enable present value with priority x in priority array, FALSE = priority x disable *)
	bNullPV				: BOOL; (* clear priority entry *)
	fPV					: REAL; (* decimal number for priority x, when input bEnablePV is TRUE *)
END_VAR
VAR_IN_OUT
	Device				: FB_BACnet_Device;
END_VAR
VAR_OUTPUT
	bReady				: BOOL;
	fPresentValue		: REAL;
	bOverridden			: BOOL;
	bOutOfService		: BOOL;
	bFault				: BOOL;
	bInAlarm			: BOOL;
	bOverRange			: BOOL;
	bUnderRange			: BOOL;
	bOtherFault			: BOOL;
	eEventState			: E_BACNETEVENTSTATE;
	bAckedTrans_ToOffNormal : BOOL;
	bAckedTrans_ToFault		: BOOL;
	bAckedTrans_ToNormal	: BOOL;
	nActivePrio			: UINT;
	tObjectID			: T_BACnet_ObjectIdentifier := 16#FFFFFFFF;
	bError				: BOOL;
	nErrorId			: UINT;
END_VAR
VAR
	_PresentValue AT%I*: REAL; 			(* ~(BACnet_PresentValue 				:		: )
								   			(BACnet_ObjectType 					: AV	: )	*)
    _PresentValue_Priority12 AT%Q*: DWORD;(* ~(BACnet_PresentValue_Priority12	:		: )	*)
	_ActivePriority AT%I*: UDINT; 		(* ~(BACnet_ActivePriority 				:		: )	*)
	_ObjectId AT%I*: DWORD;				(* ~(BACnet_ObjectIdentifier			:		: LINK) *)
	_StatusFlags AT%I*: WORD; 			(* ~(BACnet_StatusFlags 				:		: )	*)
	_EventState AT%I*: WORD;			(* ~(BACnet_EventState 					:		: )	*)
	_Reliability AT%I*: WORD;;			(* ~(BACnet_Reliability 				:		: )	*)
	_AckedTransitions AT%I*:WORD;		(* ~(BACnet_AckedTransitions			:		: ) *)
	_StatusFlagsBits : ST_BACnet_StatusFlags;
	_AckedTransBits : ST_BACnet_EventTransitionBits;
	_nUpdateCount : UDINT := 0;
END_VAR

(* update server device *)
IF (Device._nUpdateCount = _nUpdateCount) THEN
	Device();
END_IF
(* remind current number of update counter *)
_nUpdateCount := Device._nUpdateCount;

IF Device.bFirstCycle THEN
	(* first call of the server device since reboot/reset *)
	bReady := FALSE;
	_PresentValue_Priority12 := F_BACnet_RealNothing();

ELSIF (F_BACnet_GetObjType(_ObjectId) <> BACnetObjectType_AnalogValue) THEN
	(* wrong mapping / invalid object ID *)
	IF _ObjectId = 0 THEN
		nErrorId := BACnet_ERR_WRONG_MAPPING;
	ELSE
		nErrorId := BACnet_ERR_INVALID_OBJECTID;
	END_IF
	bReady := FALSE;

ELSIF (_StatusFlags < 4) THEN
	(* wrong mapping *)
	nErrorId := BACnet_ERR_WRONG_MAPPING;
	bReady := FALSE;

ELSIF Device.bOperational THEN
	(* ready state *)
	bReady := TRUE;
	nErrorId := BACnet_ERR_NO_ERROR;

	(* write into priority array *)
	_PresentValue_Priority12 := F_BACnet_RealPV(bEnablePV, bNullPV, fPV);

	(* present value *)
	fPresentValue := _PresentValue;

	(* build bit states *)
	_StatusFlagsBits := F_BACnet_StatusFlags(_StatusFlags);
	_AckedTransBits		:= F_BACnet_EventTransitionFlags(_AckedTransitions);

	(* copy states to output *)
	bOverridden := _StatusFlagsBits.overridden;
	bOutOfService := _StatusFlagsBits.out_of_service;
	bFault := _StatusFlagsBits.fault;
	bInAlarm := _StatusFlagsBits.in_alarm;
	bOverRange := (_Reliability = TO_WORD(BACnetReliability_over_range));
	bUnderRange := (_Reliability = TO_WORD(BACnetReliability_under_range));
	bOtherFault := (_Reliability = TO_WORD(BACnetReliability_unreliable_other));
	bAckedTrans_ToOffNormal := _AckedTransBits.to_offnormal;
	bAckedTrans_ToFault := _AckedTransBits.to_fault;
	bAckedTrans_ToNormal := _AckedTransBits.to_normal;
	tObjectID := _ObjectId;

	(* convert enumeration *)
	eEventState := TO_INT(_EventState);

	(* copy active priority *)
	nActivePrio := UDINT_TO_UINT(_ActivePriority);
ELSE
	(* server device not ready, reset local ready also *)
	bReady := FALSE;
	nErrorId := BACnet_ERR_OPERATIONAL;
END_IF
(* set error flag *)
bError := (nErrorId <> BACnet_ERR_NO_ERROR);

END_FUNCTION_BLOCK

// POUs/BACnet Objects/Local (Server)/Extended Process Data/FB_BACnet_Averaging_EX
FUNCTION_BLOCK FB_BACnet_Averaging_EX
VAR_IN_OUT
	Device				: FB_BACnet_Device;
END_VAR
VAR_OUTPUT
	bReady				: BOOL;
	fAverageValue		: REAL;
	fMaximumValue		: REAL;
	fMinimumValue		: REAL;
	nValidSamples		: UDINT;
	nWindowSamples		: UDINT;
	nWindowInterval		: UDINT; (* [s] *)
	tObjectID			: T_BACnet_ObjectIdentifier := 16#FFFFFFFF;
	bError				: BOOL;
	nErrorId			: UINT;
END_VAR
VAR
	_AverageValue AT%I*: REAL;			(* ~(BACnet_AverageValue	:		: )
											(BACnet_ObjectType 		: AVG	: ) *)
	_MaximumValue AT%I*: REAL;			(* ~(BACnet_MaximumValue	:		: ) *)
	_MinimumValue AT%I*: REAL;			(* ~(BACnet_MinimumValue	:		: ) *)
	_ValidSamples AT%I*: UDINT;			(* ~(BACnet_ValidSamples	:		: ) *)
	_WindowSamples AT%I*: UDINT;		(* ~(BACnet_WindowSamples	:		: ) *)
	_WindowInterval AT%I*: UDINT;		(* ~(BACnet_WindowInterval	:		: ) *)
	_ObjectId AT%I*: DWORD;				(* ~(BACnet_ObjectIdentifier:		: LINK) *)
	_nUpdateCount : UDINT := 0;
END_VAR

(* update server device *)
IF (Device._nUpdateCount = _nUpdateCount) THEN
	Device();
END_IF
(* remind current number of update counter *)
_nUpdateCount := Device._nUpdateCount;

IF Device.bFirstCycle THEN
	(* first call of the server device since reboot/reset *)
	bReady := FALSE;

ELSIF (F_BACnet_GetObjType(_ObjectId) <> BACnetObjectType_Averaging) THEN
	(* wrong mapping / invalid object ID *)
	IF _ObjectId = 0 THEN
		nErrorId := BACnet_ERR_WRONG_MAPPING;
	ELSE
		nErrorId := BACnet_ERR_INVALID_OBJECTID;
	END_IF
	bReady := FALSE;
	tObjectID := 16#FFFFFFFF;

ELSIF Device.bOperational THEN
	(* ready state *)
	bReady := TRUE;
	nErrorId := BACnet_ERR_NO_ERROR;

	(* present values *)
	fAverageValue	:= _AverageValue;
	fMaximumValue	:= _MaximumValue;
	fMinimumValue	:= _MinimumValue;
	nValidSamples	:= _ValidSamples;
	nWindowSamples	:= _WindowSamples;
	nWindowInterval	:= _WindowInterval;

	(* other states *)
	tObjectID := _ObjectId;

ELSE
	(* server device not ready, reset local ready also *)
	bReady := FALSE;
	nErrorId := BACnet_ERR_OPERATIONAL;
END_IF
(* set error flag *)
bError := (nErrorId <> BACnet_ERR_NO_ERROR);

END_FUNCTION_BLOCK

// POUs/BACnet Objects/Local (Server)/Extended Process Data/FB_BACnet_BinaryInput_EX
FUNCTION_BLOCK FB_BACnet_BinaryInput_EX
VAR_IN_OUT
	Device	: FB_BACnet_Device;
END_VAR
VAR_OUTPUT
	bReady				: BOOL;
	bPresentValue		: BOOL;
	bOverridden			: BOOL;
	bOutOfService		: BOOL;
	bFault				: BOOL;
	bInAlarm			: BOOL;
	bNoSensor			: BOOL;
	bOpenLoop			: BOOL;
	bShortedLoop		: BOOL;
	bOtherFault			: BOOL;
	eEventState			: E_BACNETEVENTSTATE;
	bAckedTrans_ToOffNormal : BOOL;
	bAckedTrans_ToFault		: BOOL;
	bAckedTrans_ToNormal	: BOOL;
	nChangeOfState		: UDINT;
	tObjectID			: T_BACnet_ObjectIdentifier := 16#FFFFFFFF;
	bError				: BOOL;
	nErrorId			: UINT;
END_VAR
VAR
	_ChangeOfStateCount AT%I*: UDINT;		(* ~(BACnet_ChangeOfStateCount	:		: ) *)
	_ObjectId AT%I*: DWORD;					(* ~(BACnet_ObjectIdentifier	:		: LINK) *)
	_PresentValue AT%I*: WORD; 				(* ~(BACnet_PresentValue 		:		: )
												(BACnet_ObjectType			:BI    	: )	*)
	_StatusFlags AT%I*: WORD; 				(* ~(BACnet_StatusFlags 		:	    : )	*)
	_EventState AT%I*: WORD; 				(* ~(BACnet_EventState 			:	    : )	*)
	_Reliability AT%I*: WORD;; 				(* ~(BACnet_Reliability 		:		: )	*)
	_AckedTransitions AT%I*:WORD;			(* ~(BACnet_AckedTransitions	:		: ) *)
	_AckedTransBits : ST_BACnet_EventTransitionBits;
	_StatusFlagsBits : ST_BACnet_StatusFlags;
	_nUpdateCount : UDINT := 0;
END_VAR

(* update server device *)
IF (Device._nUpdateCount = _nUpdateCount) THEN
	Device();
END_IF
(* remind current number of update counter *)
_nUpdateCount := Device._nUpdateCount;

(* check object type *)
IF (F_BACnet_GetObjType(_ObjectId) <> BACnetObjectType_BinaryInput) THEN
	(* wrong mapping / invalid object ID *)
	IF _ObjectId = 0 THEN
		nErrorId := BACnet_ERR_WRONG_MAPPING;
	ELSE
		nErrorId := BACnet_ERR_INVALID_OBJECTID;
	END_IF
	bReady := FALSE;

ELSIF (_StatusFlags < 4) THEN
	(* wrong mapping *)
	nErrorId := BACnet_ERR_WRONG_MAPPING;
	bReady := FALSE;

ELSIF Device.bOperational THEN
	(* ready state *)
	bReady := TRUE;
	nErrorId := BACnet_ERR_NO_ERROR;

	(* present value *)
	bPresentValue := F_BinPV_To_Bool(TO_INT(_PresentValue));

	(* build bit states *)
	_StatusFlagsBits := F_BACnet_StatusFlags(_StatusFlags);
	_AckedTransBits		:= F_BACnet_EventTransitionFlags(_AckedTransitions);

	(* copy states to output *)
	bOverridden := _StatusFlagsBits.overridden;
	bOutOfService := _StatusFlagsBits.out_of_service;
	bFault := _StatusFlagsBits.fault;
	bInAlarm := _StatusFlagsBits.in_alarm;
	bNoSensor := (_Reliability = TO_WORD(BACnetReliability_no_sensor));
	bOpenLoop := (_Reliability = TO_WORD(BACnetReliability_open_loop));
	bShortedLoop := (_Reliability = TO_WORD(BACnetReliability_shorted_loop));
	bOtherFault := (_Reliability = TO_WORD(BACnetReliability_unreliable_other));
	bAckedTrans_ToOffNormal := _AckedTransBits.to_offnormal;
	bAckedTrans_ToFault := _AckedTransBits.to_fault;
	bAckedTrans_ToNormal := _AckedTransBits.to_normal;
	tObjectID := _ObjectId;

	(* convert enumeration *)
	eEventState := TO_INT(_EventState);

	(* copy change_of_state_count *)
	nChangeOfState := _ChangeOfStateCount;
ELSE
	bReady := FALSE;
	nErrorId := BACnet_ERR_OPERATIONAL;
END_IF
(* set error flag *)
bError := (nErrorId <> BACnet_ERR_NO_ERROR);

END_FUNCTION_BLOCK

// POUs/BACnet Objects/Local (Server)/Extended Process Data/FB_BACnet_BinaryOutput_EX
FUNCTION_BLOCK FB_BACnet_BinaryOutput_EX
VAR_INPUT
	bEnablePV			: BOOL; (* enable present value with priority x in priority array, FALSE = priority x disable *)
	bNullPV				: BOOL; (* clear priority entry *)
	bPV					: BOOL; (* present value bool type *)
END_VAR
VAR_IN_OUT
	Device				: FB_BACnet_Device;
END_VAR
VAR_OUTPUT
	bReady				: BOOL;
	bPresentValue		: BOOL;
	bOverridden			: BOOL;
	bOutOfService		: BOOL;
	bFault				: BOOL;
	bInAlarm			: BOOL;
	bNoOutput			: BOOL;
	bOpenLoop			: BOOL;
	bShortedLoop		: BOOL;
	bOtherFault			: BOOL;
	eEventState			: E_BACNETEVENTSTATE;
	bAckedTrans_ToOffNormal : BOOL;
	bAckedTrans_ToFault		: BOOL;
	bAckedTrans_ToNormal	: BOOL;
	nActivePrio			: UINT;
	nChangeOfState		: UDINT;
	tObjectID			: T_BACnet_ObjectIdentifier := 16#FFFFFFFF;
	bError				: BOOL;
	nErrorId			: UINT;
END_VAR
VAR_INPUT
END_VAR
VAR
	_ActivePriority AT%I*: UDINT; 		(* ~(BACnet_ActivePriority 			:		: )	*)
	_ChangeOfStateCount AT%I*: UDINT;	(* ~(BACnet_ChangeOfStateCount		:		: ) *)
	_ObjectId AT%I*: DWORD;				(* ~(BACnet_ObjectIdentifier		:		: LINK) *)
	_PresentValue AT%I*: WORD; 			(* ~(BACnet_PresentValue 			:		: )
								   			(BACnet_ObjectType 				: BO	: )	*)
    _PresentValue_Priority12 AT%Q*: WORD;(* ~(BACnet_PresentValue_Priority12:		: )	*)
	_StatusFlags AT%I*: WORD; 			(* ~(BACnet_StatusFlags 			:		: )	*)
	_EventState AT%I*: WORD; 			(* ~(BACnet_EventState 				:		: )	*)
	_Reliability AT%I*: WORD;;			(* ~(BACnet_Reliability 			:		: )	*)
	_AckedTransitions AT%I*:WORD;		(* ~(BACnet_AckedTransitions		:		: ) *)
	_nUpdateCount : UDINT := 0;
	_AckedTransBits : ST_BACnet_EventTransitionBits;
	_StatusFlagsBits : ST_BACnet_StatusFlags;
END_VAR

(* update server device *)
IF (Device._nUpdateCount = _nUpdateCount) THEN
	Device();
END_IF
(* remind current number of update counter *)
_nUpdateCount := Device._nUpdateCount;

IF Device.bFirstCycle THEN
	(* first call of the server device since reboot/reset *)
	bReady := FALSE;
	_PresentValue_Priority12 := TO_WORD(BACnetBinaryPV_Nothing);

ELSIF (F_BACnet_GetObjType(_ObjectId) <> BACnetObjectType_BinaryOutput) THEN
	(* wrong mapping / invalid object ID *)
	IF _ObjectId = 0 THEN
		nErrorId := BACnet_ERR_WRONG_MAPPING;
	ELSE
		nErrorId := BACnet_ERR_INVALID_OBJECTID;
	END_IF
	bReady := FALSE;

ELSIF (_StatusFlags < 4) THEN
	(* wrong mapping *)
	nErrorId := BACnet_ERR_WRONG_MAPPING;
	bReady := FALSE;

ELSIF Device.bOperational THEN
	(* ready state *)
	bReady := TRUE;
	nErrorId := BACnet_ERR_NO_ERROR;

	(* write into priority array *)
	_PresentValue_Priority12 := to_word(F_Bool_To_BinPV(bEnablePV, bNullPV, bPV));

	(* present value *)
	bPresentValue := F_BinPV_To_Bool(TO_INT(_PresentValue));

	(* build bit states *)
	_StatusFlagsBits := F_BACnet_StatusFlags(_StatusFlags);
	_AckedTransBits		:= F_BACnet_EventTransitionFlags(_AckedTransitions);

	(* copy states to output *)
	bOverridden := _StatusFlagsBits.overridden;
	bOutOfService := _StatusFlagsBits.out_of_service;
	bFault := _StatusFlagsBits.fault;
	bInAlarm := _StatusFlagsBits.in_alarm;
	bNoOutput := (_Reliability = TO_WORD(BACnetReliability_no_output));
	bOpenLoop := (_Reliability = TO_WORD(BACnetReliability_open_loop));
	bShortedLoop := (_Reliability = TO_WORD(BACnetReliability_shorted_loop));
	bOtherFault := (_Reliability = TO_WORD(BACnetReliability_unreliable_other));
	bAckedTrans_ToOffNormal := _AckedTransBits.to_offnormal;
	bAckedTrans_ToFault := _AckedTransBits.to_fault;
	bAckedTrans_ToNormal := _AckedTransBits.to_normal;
	tObjectID := _ObjectId;

	(* convert enumeration *)
	eEventState := TO_INT(_EventState);

	(* copy active priority *)
	nActivePrio := UDINT_TO_UINT(_ActivePriority);

	(* copy change_of_state_count *)
	nChangeOfState := _ChangeOfStateCount;
ELSE
	(* server device not ready, reset local ready also *)
	bReady := FALSE;
	nErrorId := BACnet_ERR_OPERATIONAL;
END_IF
(* set error flag *)
bError := (nErrorId <> BACnet_ERR_NO_ERROR);

END_FUNCTION_BLOCK

// POUs/BACnet Objects/Local (Server)/Extended Process Data/FB_BACnet_BinaryValue_EX
FUNCTION_BLOCK FB_BACnet_BinaryValue_EX
VAR_INPUT
	bEnablePV			: BOOL; (* enable present value with priority x in priority array, FALSE = priority x disable *)
	bNullPV				: BOOL; (* clear priority entry *)
	bPV					: BOOL; (* present value bool type *)
END_VAR
VAR_IN_OUT
	Device				: FB_BACnet_Device;
END_VAR
VAR_OUTPUT
	bReady				: BOOL;
	bPresentValue		: BOOL;
	bOverridden			: BOOL;
	bOutOfService		: BOOL;
	bFault				: BOOL;
	bInAlarm			: BOOL;
	bOtherFault			: BOOL;
	eEventState			: E_BACNETEVENTSTATE;
	bAckedTrans_ToOffNormal : BOOL;
	bAckedTrans_ToFault		: BOOL;
	bAckedTrans_ToNormal	: BOOL;
	nActivePrio			: UINT;
	nChangeOfState		: UDINT;
	tObjectID			: T_BACnet_ObjectIdentifier := 16#FFFFFFFF;
	bError				: BOOL;
	nErrorId			: UINT;
END_VAR
VAR
	_ActivePriority AT%I*: UDINT; 		(* ~(BACnet_ActivePriority 			:		: )	*)
	_ChangeOfStateCount AT%I*: UDINT;	(* ~(BACnet_ChangeOfStateCount		:		: ) *)
	_ObjectId AT%I*: DWORD;				(* ~(BACnet_ObjectIdentifier		:		: LINK) *)
	_PresentValue AT%I*: WORD; 			(* ~(BACnet_PresentValue 			:		: )
								   			(BACnet_ObjectType 				: BV	: )	*)
    _PresentValue_Priority12 AT%Q*: WORD;(* ~(BACnet_PresentValue_Priority12:		: )	*)
	_StatusFlags AT%I*: WORD; 			(* ~(BACnet_StatusFlags 			:		: )	*)
	_EventState AT%I*: WORD; 			(* ~(BACnet_EventState 				:		: )	*)
	_Reliability AT%I*: WORD;;			(* ~(BACnet_Reliability 			:		: )	*)
	_AckedTransitions AT%I*:WORD;		(* ~(BACnet_AckedTransitions:		: 		: ) *)
	_nUpdateCount : UDINT := 0;
	_AckedTransBits : ST_BACnet_EventTransitionBits;
	_StatusFlagsBits : ST_BACnet_StatusFlags;
END_VAR

(* update server device *)
IF (Device._nUpdateCount = _nUpdateCount) THEN
	Device();
END_IF
(* remind current number of update counter *)
_nUpdateCount := Device._nUpdateCount;

IF Device.bFirstCycle THEN
	(* first call of the server device since reboot/reset *)
	bReady := FALSE;
	_PresentValue_Priority12 := TO_WORD(BACnetBinaryPV_Nothing);

ELSIF (F_BACnet_GetObjType(_ObjectId) <> BACnetObjectType_BinaryValue) THEN
	(* wrong mapping / invalid object ID *)
	IF _ObjectId = 0 THEN
		nErrorId := BACnet_ERR_WRONG_MAPPING;
	ELSE
		nErrorId := BACnet_ERR_INVALID_OBJECTID;
	END_IF
	bReady := FALSE;

ELSIF (_StatusFlags < 4) THEN
	(* wrong mapping *)
	nErrorId := BACnet_ERR_WRONG_MAPPING;
	bReady := FALSE;

ELSIF Device.bOperational THEN
	(* ready state *)
	bReady := TRUE;
	nErrorId := BACnet_ERR_NO_ERROR;

	(* write into priority array *)
	_PresentValue_Priority12 := TO_WORD(F_Bool_To_BinPV(bEnablePV, bNullPV, bPV));

	(* present value *)
	bPresentValue := F_BinPV_To_Bool(TO_INT(_PresentValue));

	(* build bit states *)
	_StatusFlagsBits := F_BACnet_StatusFlags(_StatusFlags);
	_AckedTransBits		:= F_BACnet_EventTransitionFlags(_AckedTransitions);

	(* copy states to output *)
	bOverridden := _StatusFlagsBits.overridden;
	bOutOfService := _StatusFlagsBits.out_of_service;
	bFault := _StatusFlagsBits.fault;
	bInAlarm := _StatusFlagsBits.in_alarm;
	bOtherFault := (_Reliability = TO_WORD(BACnetReliability_unreliable_other));
	bAckedTrans_ToOffNormal := _AckedTransBits.to_offnormal;
	bAckedTrans_ToFault := _AckedTransBits.to_fault;
	bAckedTrans_ToNormal := _AckedTransBits.to_normal;
	tObjectID := _ObjectId;

	(* convert enumeration *)
	eEventState := TO_INT(_EventState);

	(* copy active priority *)
	nActivePrio := UDINT_TO_UINT(_ActivePriority);

	(* copy change_of_state_count *)
	nChangeOfState := _ChangeOfStateCount;
ELSE
	(* server device not ready, reset local ready also *)
	bReady := FALSE;
	nErrorId := BACnet_ERR_OPERATIONAL;
END_IF
(* set error flag *)
bError := (nErrorId <> BACnet_ERR_NO_ERROR);

END_FUNCTION_BLOCK

// POUs/BACnet Objects/Local (Server)/Extended Process Data/FB_BACnet_Calendar_EX
FUNCTION_BLOCK FB_BACnet_Calendar_EX
VAR_IN_OUT
	Device				: FB_BACnet_Device;
END_VAR
VAR_OUTPUT
	bReady				: BOOL;
	bPresentValue		: BOOL;
	tObjectID			: T_BACnet_ObjectIdentifier := 16#FFFFFFFF;
	bError				: BOOL;
	nErrorId			: UINT;
END_VAR
VAR
	_ObjectId AT%I*: DWORD;		(* ~(BACnet_ObjectIdentifier:		: LINK) *)
	_PresentValue AT%I*: BOOL;	(* ~(BACnet_PresentValue 			:		: )
									(BACnet_ObjectType 				: CAL	: )	*)
	_nUpdateCount : UDINT := 0;
END_VAR

(* update server device *)
IF (Device._nUpdateCount = _nUpdateCount) THEN
	Device();
END_IF
(* remind current number of update counter *)
_nUpdateCount := Device._nUpdateCount;

IF (F_BACnet_GetObjType(_ObjectId) <> BACnetObjectType_Calendar) THEN
	(* wrong mapping / invalid object ID *)
	IF _ObjectId = 0 THEN
		nErrorId := BACnet_ERR_WRONG_MAPPING;
	ELSE
		nErrorId := BACnet_ERR_INVALID_OBJECTID;
	END_IF
	bReady := FALSE;
	tObjectID := 16#FFFFFFFF;

ELSIF Device.bOperational THEN
	(* ready state *)
	bReady := TRUE;
	nErrorId := BACnet_ERR_NO_ERROR;
	(* present value *)
	bPresentValue := _PresentValue;
	tObjectID := _ObjectId;
ELSE
	(* server device not ready, reset local ready also *)
	bReady := FALSE;
	nErrorId := BACnet_ERR_OPERATIONAL;
END_IF
(* set error flag *)
bError := (nErrorId <> BACnet_ERR_NO_ERROR);

END_FUNCTION_BLOCK

// POUs/BACnet Objects/Local (Server)/Extended Process Data/FB_BACnet_Command_EX
FUNCTION_BLOCK FB_BACnet_Command_EX
VAR_INPUT
	bEnablePV			: BOOL;
	nPV					: UDINT;
	bRetrigger			: BOOL; (* execute selected action on raising edge again *)
END_VAR
VAR_IN_OUT
	Device				: FB_BACnet_Device;
END_VAR
VAR_OUTPUT
	bReady				: BOOL;
	nPresentValue		: UDINT;
	bAllWritesOk		: BOOL; (* all actions in selected action list are written *)
	bInProcess			: BOOL; (* object is busy *)
	tObjectID			: T_BACnet_ObjectIdentifier := 16#FFFFFFFF;
	bError				: BOOL;
	nErrorId			: UINT;
END_VAR
VAR
	_PresentValueIn AT%I*: UDINT; 		(* ~(BACnet_PresentValue 			:		: )
								   			(BACnet_ObjectType 				: CMD	: )	*)
	_ObjectId AT%I*: DWORD;				(* ~(BACnet_ObjectIdentifier:		: LINK) *)
    _PresentValueOut AT%Q*: UDINT;		(* ~(BACnet_PresentValue	 	   	:		: )	*)
	_InProcess AT%I*: BOOL;				(* ~(BACnet_InProcess 				:		: )	*)
	_AllWritesSuccessful AT%I*: BOOL;	(* ~(BACnet_AllWritesSuccessful		:		: )	*)
	_nUpdateCount : UDINT := 0;
	_rtrigRetriggerPv : R_TRIG;
	_bRetriggerReq : BOOL;
END_VAR

(* update server device *)
IF (Device._nUpdateCount = _nUpdateCount) THEN
	Device();
END_IF
(* remind current number of update counter *)
_nUpdateCount := Device._nUpdateCount;

(* call trigger *)
_rtrigRetriggerPv(CLK:= bRetrigger, Q=> );
IF _rtrigRetriggerPv.Q THEN
	_bRetriggerReq := TRUE;
END_IF

IF Device.bFirstCycle THEN
	(* first call of the server device since reboot/reset *)
	bReady := FALSE;
	_PresentValueOut := 0;
	_bRetriggerReq := FALSE;

ELSIF (F_BACnet_GetObjType(_ObjectId) <> BACnetObjectType_Command) THEN
	(* wrong mapping / invalid object ID *)
	IF _ObjectId = 0 THEN
		nErrorId := BACnet_ERR_WRONG_MAPPING;
	ELSE
		nErrorId := BACnet_ERR_INVALID_OBJECTID;
	END_IF
	bReady := FALSE;
	tObjectID := 16#FFFFFFFF;
	_bRetriggerReq := FALSE;

ELSIF Device.bOperational THEN
	(* object ID *)
	tObjectID := _ObjectId;
	(* ready state *)
	bReady := TRUE;
	nErrorId := BACnet_ERR_NO_ERROR;
	(* activities *)
	bAllWritesOk := _AllWritesSuccessful;
	bInProcess := _InProcess;
	(* present value from BACnet *)
	nPresentValue := _PresentValueIn;
	(* present value to BACnet *)
	IF bEnablePV THEN
		IF (NOT bInProcess) THEN
			IF _bRetriggerReq THEN
				(* trigger action list *)
				_PresentValueOut := 0;
			ELSE
				(* set present value *)
				_PresentValueOut := nPV;
			END_IF
			_bRetriggerReq := FALSE;
		END_IF
	ELSE
		(* deactivate mapped present value --> other objects can write to property *)
		_PresentValueOut := 16#0;
		_bRetriggerReq := FALSE;
	END_IF
ELSE
	(* server device not ready, reset local ready also *)
	bReady := FALSE;
	nErrorId := BACnet_ERR_OPERATIONAL;
	_bRetriggerReq := FALSE;
END_IF
(* set error flag *)
bError := (nErrorId <> BACnet_ERR_NO_ERROR);

END_FUNCTION_BLOCK

// POUs/BACnet Objects/Local (Server)/Extended Process Data/FB_BACnet_EventEnrollment_EX
FUNCTION_BLOCK FB_BACnet_EventEnrollment_EX
VAR_IN_OUT
	Device				: FB_BACnet_Device;
END_VAR
VAR_OUTPUT
	bReady				: BOOL;
	eEventState			: E_BACNETEVENTSTATE;
	bEventEnable_ToOffNormal: BOOL;
	bEventEnable_ToFault: BOOL;
	bEventEnable_ToNormal: BOOL;
	bAckedTrans_ToOffNormal: BOOL;
	bAckedTrans_ToFault	: BOOL;
	bAckedTrans_ToNormal: BOOL;
	tObjectID			: T_BACnet_ObjectIdentifier := 16#FFFFFFFF;
	bError				: BOOL;
	nErrorId			: UINT;
END_VAR
VAR
	_ObjectId AT%I*: DWORD;			(* ~(BACnet_ObjectIdentifier	:		: LINK) *)
	_EventState AT%I*: WORD; 		(* ~(BACnet_EventState 			:		: )
										(BACnet_ObjectType			: EE	: )	*)
	_AckedTransitions AT%I*: WORD; 	(* ~(BACnet_AckedTransitions 	:		: )	*)
	_EventEnable AT%I*: WORD; 		(* ~(BACnet_EventEnable		 	:		: )	*)
	_EventTransBits : ST_BACnet_EventTransitionBits;
	_nUpdateCount : UDINT := 0;
END_VAR

(* update server device *)
IF (Device._nUpdateCount = _nUpdateCount) THEN
	Device();
END_IF
(* remind current number of update counter *)
_nUpdateCount := Device._nUpdateCount;

(* check BitString format *)
IF (F_BACnet_GetObjType(_ObjectId) <> BACnetObjectType_EventEnrollment) THEN
	(* wrong mapping / invalid object ID *)
	IF _ObjectId = 0 THEN
		nErrorId := BACnet_ERR_WRONG_MAPPING;
	ELSE
		nErrorId := BACnet_ERR_INVALID_OBJECTID;
	END_IF
	bReady := FALSE;
	tObjectID := 16#FFFFFFFF;

ELSIF (_AckedTransitions < 5) THEN
	(* wrong mapping *)
	nErrorId := BACnet_ERR_WRONG_MAPPING;
	bReady := FALSE;

ELSIF Device.bOperational THEN
	(* ready state *)
	bReady := TRUE;
	nErrorId := BACnet_ERR_NO_ERROR;

	(* copy states *)
	_EventTransBits			:= F_BACnet_EventTransitionFlags(_AckedTransitions);
	bAckedTrans_ToOffNormal	:= _EventTransBits.to_offnormal;
	bAckedTrans_ToFault		:= _EventTransBits.to_fault;
	bAckedTrans_ToNormal	:= _EventTransBits.to_normal;
	_EventTransBits			:= F_BACnet_EventTransitionFlags(_EventEnable);
	bEventEnable_ToOffNormal:= _EventTransBits.to_offnormal;
	bEventEnable_ToFault	:= _EventTransBits.to_fault;
	bEventEnable_ToNormal	:= _EventTransBits.to_normal;
	eEventState				:= TO_INT(_EventState);
	tObjectID			:= F_BACnet_GetObjInstance(_ObjectId);

ELSE
	bReady := FALSE;
	nErrorId := BACnet_ERR_OPERATIONAL;
END_IF
(* set error flag *)
bError := (nErrorId <> BACnet_ERR_NO_ERROR);

END_FUNCTION_BLOCK

// POUs/BACnet Objects/Local (Server)/Extended Process Data/FB_BACnet_File_EX
FUNCTION_BLOCK FB_BACnet_File_EX
VAR_IN_OUT
	Device				: FB_BACnet_Device;
END_VAR
VAR_OUTPUT
	bReady				: BOOL;
	nFileSize			: UDINT;
	tObjectID			: T_BACnet_ObjectIdentifier := 16#FFFFFFFF;
	bError				: BOOL;
	nErrorId			: UINT;
END_VAR
VAR
	_FileSize 			AT%I*: UDINT; 	(* ~(BACnet_FileSize 		:		: )
					   						(BACnet_ObjectType 		: FILE	: )	*)
	_ObjectId AT%I*: DWORD;				(* ~(BACnet_ObjectIdentifier:		: LINK) *)
	_nUpdateCount		: UDINT := 0;
END_VAR

(* update server device *)
IF (Device._nUpdateCount = _nUpdateCount) THEN
	Device();
END_IF
(* remind current number of update counter *)
_nUpdateCount := Device._nUpdateCount;

IF (F_BACnet_GetObjType(_ObjectId) <> BACnetObjectType_File) THEN
	(* wrong mapping / invalid object ID *)
	IF _ObjectId = 0 THEN
		nErrorId := BACnet_ERR_WRONG_MAPPING;
	ELSE
		nErrorId := BACnet_ERR_INVALID_OBJECTID;
	END_IF
	bReady := FALSE;
	tObjectID := 16#FFFFFFFF;

ELSIF Device.bOperational THEN
	(* ready state *)
	bReady := TRUE;
	nErrorId := BACnet_ERR_NO_ERROR;
	nFileSize := _FileSize;
	tObjectID := _ObjectId;

ELSE
	(* server device not ready, reset local ready also *)
	bReady := FALSE;
	nErrorId := BACnet_ERR_OPERATIONAL;
END_IF
(* set error flag *)
bError := (nErrorId <> BACnet_ERR_NO_ERROR);

END_FUNCTION_BLOCK

// POUs/BACnet Objects/Local (Server)/Extended Process Data/FB_BACnet_Group_EX
FUNCTION_BLOCK FB_BACnet_Group_EX
VAR_IN_OUT
	Device				: FB_BACnet_Device;
END_VAR
VAR_OUTPUT
	bReady				: BOOL;
	tObjectID			: T_BACnet_ObjectIdentifier := 16#FFFFFFFF;
	bError				: BOOL;
	nErrorId			: UINT;
END_VAR
VAR
	_ObjectId AT%I*: DWORD;		(* ~(BACnet_ObjectIdentifier:		: LINK)
									(BACNET_OBJECTTYPE		: GROUP : ) *)
	_nUpdateCount : UDINT := 0;
END_VAR

(* update server device *)
IF (Device._nUpdateCount = _nUpdateCount) THEN
	Device();
END_IF
(* remind current number of update counter *)
_nUpdateCount := Device._nUpdateCount;

IF (F_BACnet_GetObjType(_ObjectId) <> BACnetObjectType_Group) THEN
	(* wrong mapping / invalid object ID *)
	IF _ObjectId = 0 THEN
		nErrorId := BACnet_ERR_WRONG_MAPPING;
	ELSE
		nErrorId := BACnet_ERR_INVALID_OBJECTID;
	END_IF
	bReady := FALSE;
	tObjectID := 16#FFFFFFFF;

ELSIF Device.bOperational THEN
	(* ready state *)
	bReady := TRUE;
	nErrorId := BACnet_ERR_NO_ERROR;
	tObjectID := _ObjectId;
ELSE
	(* server device not ready, reset local ready also *)
	bReady := FALSE;
	nErrorId := BACnet_ERR_OPERATIONAL;
END_IF
(* set error flag *)
bError := (nErrorId <> BACnet_ERR_NO_ERROR);

END_FUNCTION_BLOCK

// POUs/BACnet Objects/Local (Server)/Extended Process Data/FB_BACnet_Loop_EX
FUNCTION_BLOCK FB_BACnet_Loop_EX
VAR_INPUT
	bAutoTuning			: BOOL; (* Start autotuning of PID controller *)
	tTuningTimeout		: TIME := T#15m; (* Maximum runtime of tuning procedure [ms] *)
	eTuningMode			: E_BACNETPIDTUNINGMODE := BACnetPIDTuningMode_PI; (* optimize default PI controller *)
	fAccLimit			: REAL := 0.0; (* Setpoint acceleration limit positive and negative [1/s] *)
END_VAR
VAR_IN_OUT
	Device				: FB_BACnet_Device;
END_VAR
VAR_OUTPUT
	bReady				: BOOL;
	bTuningActive		: BOOL;
	bTuningWaitPV		: BOOL;
	bTuningWaitCV		: BOOL;
	bTuningDone			: BOOL;
	bTuningAborted		: BOOL;
	fSetPoint			: REAL;
	fControlledValue	: REAL;
	fPresentValue		: REAL;
	fPropBand			: REAL; (* controller output in range of -100...100% in relation to Min.-/Max.-output *)
	bOverridden			: BOOL;
	bOutOfService		: BOOL;
	bFault				: BOOL;
	bInAlarm			: BOOL;
	bOpenLoop			: BOOL;
	bCommFailure		: BOOL;
	bOtherFault			: BOOL;
	eEventState			: E_BACNETEVENTSTATE;
	bAckedTrans_ToOffNormal : BOOL;
	bAckedTrans_ToFault		: BOOL;
	bAckedTrans_ToNormal	: BOOL;
	tObjectID			: T_BACnet_ObjectIdentifier := 16#FFFFFFFF;
	bError				: BOOL;
	nErrorId			: UINT;
	eMode				: E_BACNETLOOPMODE; (* mode is detected by the unit of property Integral_Constant and Derivative_Constant (Time_seconds = BACnetLoopMode_Standard) *)
END_VAR
VAR
	_ControlledVariableValue AT%I*: REAL;	(* ~(BACnet_ControlledVariableValue :		: )
												(BACnet_ObjectType				: LOOP	: )	*)
	_Setpoint AT%I*:REAL;					(* ~(BACnet_Setpoint				:		: )	*)
	_ProportionalConstant AT%I*:REAL;		(* ~(BACnet_ProportionalConstant	:		: )	*)
	_IntegralConstant AT%I*:REAL;			(* ~(BACnet_IntegralConstant	 	:		: )	*)
	_DerivativeConstant AT%I*:REAL;			(* ~(BACnet_DerivativeConstant	 	:		: )	*)
	_MaximumOutput AT%I*:REAL;				(* ~(BACnet_MaximumOutput			:		: )	*)
	_MinimumOutput AT%I*:REAL;				(* ~(BACnet_MinimumOutput			:		: )	*)
	_Bias AT%I*:REAL;						(* ~(BACnet_Bias					:		: )	*)
	_PresentValueI AT%I*: REAL; 			(* ~(BACnet_PresentValue 			: 		: )	*)
	_Deadband AT%I*: REAL; 					(* ~(BACnet_Deadband	 			: 		: )	*)
	_ObjectId AT%I*: DWORD;					(* ~(BACnet_ObjectIdentifier		:		: LINK) *)
	_StatusFlags AT%I*: WORD; 				(* ~(BACnet_StatusFlags 			: 		: )	*)
	_AckedTransitions AT%I*:WORD;			(* ~(BACnet_AckedTransitions		:		: ) *)
	_EventState AT%I*: WORD; 				(* ~(BACnet_EventState 				:		: )	*)
	_Reliability AT%I*: WORD;				(* ~(BACNET_RELIABILITY 			:		: )	*)
	_ControlAction AT%I*:E_BACNETACTION;	(* ~(BACNET_ACTION				 	:		: )	*)
	_PropConstantUnits AT%I*:E_BACNETUNIT;	(* ~(BACnet_ProportionalConstantUnits:	Other_no_units	: WRITEPROTECT) *)
	_IntegralConstUnits AT%I*:E_BACNETUNIT;	(* ~(BACnet_IntegralConstantUnits	:	Other_no_units	: WRITEPROTECT) *)
	_DerivativeConstUnits AT%I*:E_BACNETUNIT;(*~(BACnet_DerivativeConstantUnits	:	Other_no_units	: WRITEPROTECT) *)
	_PresentValueQ AT%Q*: REAL;				(* ~(BACnet_PresentValue	 		:		: )	*)
	_AckedTransBits : ST_BACnet_EventTransitionBits;
	_StatusFlagsBits : ST_BACnet_StatusFlags;

	_sysTime	: GETCPUCOUNTER;
	_Time		: T_LARGE_INTEGER;
	_TimeOld	: T_LARGE_INTEGER;
	_cycleTime	: REAL;
	_PidControl : FB_BACnet_PidControl;
	_AutoTuning : _FB_BACnet_PidTune;
	_iTuning	: INT;
	_WriteProp	: FB_BACnet_WriteProp;
	_fbAccLimit : FB_BACnet_AccLimit;
	_nUpdateCount : UDINT := 0;

	_fTuneKp	: REAL;
	_fTuneKi	: REAL;
	_fTuneKd	: REAL;

END_VAR

(* update server device *)
IF (Device._nUpdateCount = _nUpdateCount) THEN
	Device();
END_IF
(* remind current number of update counter *)
_nUpdateCount := Device._nUpdateCount;

(* determine cycle time *)
_TimeOld := _Time;
_sysTime(cpuCntLoDW=> _Time.dwLowPart, cpuCntHiDW=> _Time.dwHighPart);
_cycleTime := _F_BACnet_SysTimeDiff(In1:=_Time, In2:=_TimeOld);

(* check BitString format of StatusFlags --> if StatusFlags are less than 4, object isn't linked correctly *)
IF (F_BACnet_GetObjType(_ObjectId) <> BACnetObjectType_Loop) THEN
	(* wrong mapping / invalid object ID *)
	IF _ObjectId = 0 THEN
		nErrorId := BACnet_ERR_WRONG_MAPPING;
	ELSE
		nErrorId := BACnet_ERR_INVALID_OBJECTID;
	END_IF
	bReady := FALSE;
	tObjectID := 16#FFFFFFFF;

ELSIF (_StatusFlags < 4) THEN
	(* wrong mapping *)
	nErrorId := BACnet_ERR_WRONG_MAPPING;
	bReady := FALSE;

ELSIF Device.bOperational THEN
	(* ready state *)
	bReady := TRUE;
	nErrorId := BACnet_ERR_NO_ERROR;

	(* decode status flags *)
	_StatusFlagsBits := F_BACnet_StatusFlags(_StatusFlags);
	_AckedTransBits	:= F_BACnet_EventTransitionFlags(_AckedTransitions);

	(* copy states to output *)
	bOverridden := _StatusFlagsBits.overridden;
	bOutOfService := _StatusFlagsBits.out_of_service;
	bFault := _StatusFlagsBits.fault;
	bInAlarm := _StatusFlagsBits.in_alarm;
	bOpenLoop := (_Reliability = TO_WORD(BACnetReliability_open_loop));
	bCommFailure := (_Reliability = TO_WORD(BACnetReliability_communication_failure));
	bOtherFault := (_Reliability = TO_WORD(BACnetReliability_unreliable_other));
	bAckedTrans_ToOffNormal := _AckedTransBits.to_offnormal;
	bAckedTrans_ToFault := _AckedTransBits.to_fault;
	bAckedTrans_ToNormal := _AckedTransBits.to_normal;
	tObjectID := _ObjectId;
	eEventState := TO_INT(_EventState);

	(* check PID mode *)
	IF		(_IntegralConstUnits = BACnetUnit_Time_seconds)
		AND	(_DerivativeConstUnits = BACnetUnit_Time_seconds)
		AND (_PropConstantUnits = BACnetUnit_Other_no_units)
	THEN
		(* both are time_seconds *)
		eMode := BACnetLoopMode_Standard;
	ELSIF	(_IntegralConstUnits <> BACnetUnit_Time_seconds)
		AND	(_DerivativeConstUnits <> BACnetUnit_Time_seconds)
		AND (_PropConstantUnits = BACnetUnit_Other_no_units)
		(* both are not time_seconds *)
	THEN
		eMode := BACnetLoopMode_Ideal;
	ELSE
		(* unknown settings - stop controller *)
		eMode := BACnetLoopMode_None;
	END_IF

	(* check if auto tuning is active *)
	IF bTuningActive THEN
		_PidControl.bReset			:= TRUE;

	(* check reliability and mode *)
	ELSIF		_Reliability <> TO_WORD(BACnetReliability_no_fault_detected)
		OR	(eMode = BACnetLoopMode_None)
	THEN
		_PidControl.bReset			:= TRUE;

	(* is set out of service? *)
	ELSIF _StatusFlagsBits.out_of_service THEN
		_PidControl.bReset			:= TRUE;

	(* decide the control action (direct or reverse) *)
	ELSIF _ControlAction = BACnetAction_direct THEN
		_PidControl.bReset			:= FALSE;
		_PidControl.fPresentValue	:= _ControlledVariableValue;
		_PidControl.fSetpoint		:= _Setpoint;

	ELSIF _ControlAction = BACnetAction_reverse THEN
		_PidControl.bReset			:= FALSE;
		_PidControl.fPresentValue	:= _Setpoint;
		_PidControl.fSetpoint		:= _ControlledVariableValue;

	ELSE
		(* unknown action *)
		_PidControl.bReset			:= TRUE;
	END_IF

	(* set parameter depending on mode *)
	CASE eMode OF
		BACnetLoopMode_Ideal:
			_PidControl.fKp := _ProportionalConstant;
			_PidControl.fKi	:= _IntegralConstant;
			_PidControl.fKd	:= _DerivativeConstant;
		BACnetLoopMode_Standard:
			(* Kp = Kp *)
			_PidControl.fKp := _ProportionalConstant;
			(* Ki = Kp / Ti *)
			IF (_IntegralConstant <> 0.0) THEN
				_PidControl.fKi	:= _ProportionalConstant / _IntegralConstant;
			ELSE
				_PidControl.fKi	:= 0.0;
			END_IF
			(* Kd = Kp * Td *)
			_PidControl.fKd	:= _ProportionalConstant * _DerivativeConstant;
	END_CASE

	(* call PID control function block *)
	_PidControl(
		fCtrlCycleTime	:= _cycleTime,
		fBias			:= _Bias,
		fTp				:= -1.0,
		fMaxOutput		:= _MaximumOutput,
		fMinOutput		:= _MinimumOutput,
		nErrorStatus	=>
	);
	IF (_iTuning < 10) THEN
		_fbAccLimit.X := _PidControl.fY;
	END_IF

	(* set other outputs *)
	fSetPoint := _Setpoint;
	fPresentValue := _PresentValueI;
	fControlledValue := _ControlledVariableValue;
ELSE
	(* server device not ready, reset local ready also *)
	bReady := FALSE;
	nErrorId := BACnet_ERR_OPERATIONAL;
END_IF

(* write controller settings *)
_WriteProp.BACnetDevicePort:= Device.stAdsConn.nAmsPort;
_WriteProp.sNetId		:= Device.stAdsConn.sAmsNetId;
_WriteProp.ObjectType	:= BACnetObjectType_Loop;
_WriteProp.ObjectInstance:= F_BACnet_GetObjInstance(_ObjectId);

(* Autotuning function *)
CASE _iTuning OF
	0: (* Idle *)
		IF		bReady						(* object ready *)
			AND	(NOT _PidControl.bReset)	(* PID controller ready *)
			AND (tTuningTimeout > t#0ms)	(* timeout valid *)
			AND bAutoTuning					(* start flag *)
		THEN
			_iTuning := 5;
		END_IF
		_AutoTuning.bStart := FALSE;

	5:
		(* present_value low *)
		IF (_PresentValueI <= ((_MaximumOutput + _MinimumOutput) / 2.0) + _Bias) THEN
			_iTuning := 10;
		ELSIF (NOT bAutoTuning) THEN
			_iTuning := 0;
		END_IF

	10: (* setup *)
		_AutoTuning.fSetY	:= _MaximumOutput;
		_AutoTuning.tTimeout:= tTuningTimeout;
		_AutoTuning.fMinY	:= _MinimumOutput;
		_AutoTuning.fMaxY	:= _MaximumOutput;
		_AutoTuning.fDeadband:= _Deadband;
		_AutoTuning.eMode	:= eTuningMode;
		_iTuning := 20;

	20: (* wait busy *)
		_AutoTuning.bStart := TRUE;
		IF _AutoTuning.bAborted THEN
			_iTuning := 200;
		ELSIF _AutoTuning.bBusy THEN
			_iTuning := 30;
		END_IF

	30: (* wait done *)
		IF _AutoTuning.bAborted THEN
			_iTuning := 200;
		ELSIF _AutoTuning.bDone THEN
			_iTuning := 40;
		END_IF

	40: (* write properties *)
		IF Device.stAdsConn.bValid THEN
			_iTuning := 41;
			_WriteProp(bExecute := FALSE);
			IF (eMode = BACnetLoopMode_Ideal) THEN
				_fTuneKp := _AutoTuning.fPID_Kp;
				_fTuneKi := _AutoTuning.fPID_Ki;
				_fTuneKd := _AutoTuning.fPID_Kd;
			ELSE
				_fTuneKp := _AutoTuning.fPID_Kp;
				IF (_AutoTuning.fPID_Ki <> 0.0) THEN
					_fTuneKi := _fTuneKp / _AutoTuning.fPID_Ki;
				ELSE
					_fTuneKi := 0.0;
				END_IF
				IF (_fTuneKp <> 0.0) THEN
					_fTuneKd := _AutoTuning.fPID_Kd / _fTuneKp;
				ELSE
					_fTuneKd := 0.0;
				END_IF
			END_IF
		ELSE
			_iTuning := 200;
		END_IF

	41: (* write Kp *)
		_WriteProp.DataType	:= BACnetDataType_Real;
		_WriteProp.ptrValue	:= ADR(_fTuneKp);
		_WriteProp.nLenValue:= SIZEOF(_fTuneKp);
		_WriteProp(
			bExecute := TRUE,
			PropertyID := BACnetPropertyIdentifier_ProportionalConstant);
		IF (NOT _WriteProp.bBusy) THEN
			IF (_WriteProp.bError) THEN
				_iTuning := 200;
			ELSE
				_iTuning := 42;
			END_IF
			_WriteProp(bExecute := FALSE);
		END_IF

	42: (* write Ki *)
		_WriteProp.DataType	:= BACnetDataType_Real;
		_WriteProp.ptrValue	:= ADR(_fTuneKi);
		_WriteProp.nLenValue:= SIZEOF(_fTuneKi);
		_WriteProp(
			bExecute := TRUE,
			PropertyID := BACnetPropertyIdentifier_IntegralConstant);
		IF (NOT _WriteProp.bBusy) THEN
			IF (_WriteProp.bError) THEN
				_iTuning := 200;
			ELSE
				_iTuning := 43;
			END_IF
			_WriteProp(bExecute := FALSE);
		END_IF

	43: (* write Kd *)
		_WriteProp.DataType	:= BACnetDataType_Real;
		_WriteProp.ptrValue	:= ADR(_fTuneKd);
		_WriteProp.nLenValue:= SIZEOF(_fTuneKd);
		_WriteProp(
			bExecute := TRUE,
			PropertyID := BACnetPropertyIdentifier_DerivativeConstant);
		IF (NOT _WriteProp.bBusy) THEN
			IF (_WriteProp.bError) THEN
				_iTuning := 200;
			ELSE
				_iTuning := 44;
			END_IF
			_WriteProp(bExecute := FALSE);
		END_IF

	44: (* write Action *)
		_WriteProp.DataType	:= BACnetDataType_Enumerated;
		_WriteProp.ptrValue	:= ADR(_AutoTuning.eAction);
		_WriteProp.nLenValue:= SIZEOF(_AutoTuning.eAction);
		_WriteProp(
			bExecute := TRUE,
			PropertyID := BACnetPropertyIdentifier_Action);
		IF (NOT _WriteProp.bBusy) THEN
			IF (_WriteProp.bError) THEN
				_iTuning := 200;
			ELSE
				_iTuning := 100;
			END_IF
			_WriteProp(bExecute := FALSE);
		END_IF


	100: (* done *)
		IF NOT bAutoTuning THEN
			_iTuning := 0;
		END_IF

	200: (* aborted *)
		IF NOT bAutoTuning THEN
			_iTuning := 0;
		END_IF

END_CASE

(* call auto tuning function block *)
_AutoTuning(
	bStart	:= ,
	bStop	:=	_StatusFlagsBits.out_of_service
			OR	_Reliability <> TO_WORD(BACnetReliability_no_fault_detected),
	fSetY	:= ,
	fDeadband	:= ,
	fX		:= _ControlledVariableValue,
	tTimeout:= ,
	fMinY	:= ,
	fMaxY	:= ,
	fCycleTime := _cycleTime,
	fY		:= _fbAccLimit.X,
	fPID_Kp	=> ,
	fPID_Ki	=> ,
	fPID_Kd	=> ,
	eAction => ,
	bSetY	=> ,
	bWaitY	=> ,
	bWaitX	=> ,
	bReady	=> ,
	bBusy	=> ,
	bDone	=> ,
	bAborted=> bTuningAborted,
	bTimeout=> );

(* set auto tuning state *)
bTuningWaitPV	:= (_iTuning = 5);
bTuningWaitCV	:= (_iTuning > 5 AND _iTuning <= 30);
bTuningAborted	:= (_iTuning = 200);
bTuningActive	:= (_iTuning > 0) AND (NOT bTuningAborted);
bTuningDone		:= (_iTuning = 100);
(* set error info *)
IF (bTuningActive OR bTuningAborted) THEN
	IF (NOT Device.stAdsConn.bValid) THEN
		nErrorId	:= BACnet_ERR_INVALID_ADS_CONN;
	ELSIF _WriteProp.bError THEN
		nErrorId	:= BACnet_ERR_ADS_Write;
	END_IF
END_IF

(* limit present value *)
_fbAccLimit(
	X	:= ,
	Amax:= fAccLimit,
	Tcycle:= _cycleTime,
	Y	=> _PresentValueQ,
	A	=> );

(* calculate proportional band *)
IF (_MaximumOutput > 0.0) AND (_MinimumOutput >= 0.0) THEN
	fPropBand := ((_PresentValueQ - _MinimumOutput) / (_MaximumOutput - _MinimumOutput)) * 100.0;
ELSIF (_MaximumOutput <= 0.0) AND (_MinimumOutput < 0.0) THEN
	fPropBand := ((_PresentValueQ - _MaximumOutput) / (_MaximumOutput - _MinimumOutput)) * 100.0;
ELSIF (_PresentValueQ > 0.0) AND (_MaximumOutput > 0.0) THEN
	fPropBand := (_PresentValueQ / _MaximumOutput) * 100.0;
ELSIF (_PresentValueQ < 0.0) AND (_MinimumOutput < 0.0) THEN
	fPropBand := (_PresentValueQ / _MinimumOutput) * -100.0;
ELSE
	fPropBand := 0.0;
END_IF

(* set error flag *)
bError := (nErrorId <> BACnet_ERR_NO_ERROR);

END_FUNCTION_BLOCK

// POUs/BACnet Objects/Local (Server)/Extended Process Data/FB_BACnet_MultiStateInput_EX
FUNCTION_BLOCK FB_BACnet_MultiStateInput_EX
VAR_IN_OUT
	Device				: FB_BACnet_Device;
END_VAR
VAR_OUTPUT
	bReady				: BOOL;
	nPresentValue		: UDINT;
	bOverridden			: BOOL;
	bOutOfService		: BOOL;
	bFault				: BOOL;
	bInAlarm			: BOOL;
	bOverRange			: BOOL;
	bUnderRange			: BOOL;
	bNoSensor			: BOOL;
	bOpenLoop			: BOOL;
	bShortedLoop		: BOOL;
	bMultiStateFault	: BOOL;
	bOtherFault			: BOOL;
	eEventState			: E_BACNETEVENTSTATE;
	bAckedTrans_ToOffNormal : BOOL;
	bAckedTrans_ToFault		: BOOL;
	bAckedTrans_ToNormal	: BOOL;
	nNbrOfStates		: UDINT;
	tObjectID			: T_BACnet_ObjectIdentifier := 16#FFFFFFFF;
	bError				: BOOL;
	nErrorId			: UINT;
END_VAR
VAR
	_PresentValue AT%I*: UDINT; 		(* ~(BACnet_PresentValue 	:		: )
								   			(BACnet_ObjectType 		: MI	: )	*)
	_NumberOfStates AT%I*: UDINT;		(* ~(BACnet_NumberOfStates	:		: )	*)
	_ObjectId AT%I*: DWORD;				(* ~(BACnet_ObjectIdentifier:		: LINK) *)
	_StatusFlags AT%I*: WORD; 			(* ~(BACnet_StatusFlags 	:		: )	*)
	_EventState AT%I*: WORD; 			(* ~(BACnet_EventState 		:		: )	*)
	_Reliability AT%I*: WORD;; 			(* ~(BACnet_Reliability 	:		: )	*)
	_AckedTransitions AT%I*:WORD;		(* ~(BACnet_AckedTransitions:		: ) *)
	_AckedTransBits : ST_BACnet_EventTransitionBits;
	_nUpdateCount : UDINT := 0;
	_StatusFlagsBits : ST_BACnet_StatusFlags;
END_VAR

(* update server device *)
IF (Device._nUpdateCount = _nUpdateCount) THEN
	Device();
END_IF
(* remind current number of update counter *)
_nUpdateCount := Device._nUpdateCount;

(* check object type *)
IF (F_BACnet_GetObjType(_ObjectId) <> BACnetObjectType_MultiStateInput) THEN
	(* wrong mapping / invalid object ID *)
	IF _ObjectId = 0 THEN
		nErrorId := BACnet_ERR_WRONG_MAPPING;
	ELSE
		nErrorId := BACnet_ERR_INVALID_OBJECTID;
	END_IF
	bReady := FALSE;

ELSIF (_StatusFlags < 4) THEN
	(* wrong mapping *)
	nErrorId := BACnet_ERR_WRONG_MAPPING;
	bReady := FALSE;

ELSIF Device.bOperational THEN
	(* ready state *)
	bReady := TRUE;
	nErrorId := BACnet_ERR_NO_ERROR;

	(* present value *)
	nPresentValue := _PresentValue;

	(* build bit states *)
	_StatusFlagsBits := F_BACnet_StatusFlags(_StatusFlags);
	_AckedTransBits		:= F_BACnet_EventTransitionFlags(_AckedTransitions);

	(* copy states to output *)
	bOverridden := _StatusFlagsBits.overridden;
	bOutOfService := _StatusFlagsBits.out_of_service;
	bFault := _StatusFlagsBits.fault;
	bInAlarm := _StatusFlagsBits.in_alarm;
	bOverRange := (_Reliability = TO_WORD(BACnetReliability_over_range));
	bUnderRange := (_Reliability = TO_WORD(BACnetReliability_under_range));
	bNoSensor := (_Reliability = TO_WORD(BACnetReliability_no_sensor));
	bOpenLoop := (_Reliability = TO_WORD(BACnetReliability_open_loop));
	bShortedLoop := (_Reliability = TO_WORD(BACnetReliability_shorted_loop));
	bMultiStateFault := (_Reliability = TO_WORD(BACnetReliability_multi_state_fault));
	bOtherFault := (_Reliability = TO_WORD(BACnetReliability_unreliable_other));
	bAckedTrans_ToOffNormal := _AckedTransBits.to_offnormal;
	bAckedTrans_ToFault := _AckedTransBits.to_fault;
	bAckedTrans_ToNormal := _AckedTransBits.to_normal;
	tObjectID := _ObjectId;

	(* convert enumeration *)
	eEventState := TO_INT(_EventState);

	(* number of states *)
	nNbrOfStates := _NumberOfStates;

ELSE
	(* server device not ready, reset local ready also *)
	bReady := FALSE;
	nErrorId := BACnet_ERR_OPERATIONAL;
END_IF
(* set error flag *)
bError := (nErrorId <> BACnet_ERR_NO_ERROR);

END_FUNCTION_BLOCK

// POUs/BACnet Objects/Local (Server)/Extended Process Data/FB_BACnet_MultiStateOutput_EX
FUNCTION_BLOCK FB_BACnet_MultiStateOutput_EX
VAR_INPUT
	bEnablePV			: BOOL; (* enable present value with priority x in priority array, FALSE = priority x disable *)
	bNullPV				: BOOL; (* clear priority entry *)
	nPV					: UDINT; (* number for priority x, when input bEnablePV is TRUE *)
END_VAR
VAR_IN_OUT
	Device				: FB_BACnet_Device;
END_VAR
VAR_OUTPUT
	bReady				: BOOL;
	nPresentValue		: UDINT;
	bOverridden			: BOOL;
	bOutOfService		: BOOL;
	bFault				: BOOL;
	bInAlarm			: BOOL;
	bNoOutput			: BOOL;
	bOpenLoop			: BOOL;
	bShortedLoop		: BOOL;
	bOtherFault			: BOOL;
	eEventState			: E_BACNETEVENTSTATE;
	bAckedTrans_ToOffNormal : BOOL;
	bAckedTrans_ToFault		: BOOL;
	bAckedTrans_ToNormal	: BOOL;
	nActivePrio			: UINT;
	nNbrOfStates		: UDINT;
	tObjectID			: T_BACnet_ObjectIdentifier := 16#FFFFFFFF;
	bError				: BOOL;
	nErrorId			: UINT;
END_VAR
VAR
	_PresentValue AT%I*: UDINT; 			(* ~(BACnet_PresentValue 		:		: )
								   				(BACnet_ObjectType			: MO	: )	*)
    _PresentValue_Priority12 AT%Q*: UDINT;	(* ~(BACnet_PresentValue_Priority12		:		: )	*)
	_ActivePriority AT%I*: UDINT; 			(* ~(BACnet_ActivePriority 		:		: )	*)
	_NumberOfStates AT%I*: UDINT;			(* ~(BACnet_NumberOfStates		:		: )	*)
	_ObjectId AT%I*: DWORD;					(* ~(BACnet_ObjectIdentifier	:		: LINK) *)
	_StatusFlags AT%I*: WORD; 				(* ~(BACnet_StatusFlags			:		: )	*)
	_EventState AT%I*: WORD;				(* ~(BACnet_EventState			:		: )	*)
	_Reliability AT%I*: WORD;; 				(* ~(BACnet_Reliability			:		: )	*)
	_AckedTransitions AT%I*:WORD;			(* ~(BACnet_AckedTransitions	:		: ) *)
	_AckedTransBits : ST_BACnet_EventTransitionBits;
	_nUpdateCount : UDINT := 0;
	_StatusFlagsBits : ST_BACnet_StatusFlags;
END_VAR

(* update server device *)
IF (Device._nUpdateCount = _nUpdateCount) THEN
	Device();
END_IF
(* remind current number of update counter *)
_nUpdateCount := Device._nUpdateCount;

IF Device.bFirstCycle THEN
	(* first call of the server device since reboot/reset *)
	bReady := FALSE;
	_PresentValue_Priority12 := 16#FFFFFFFF;

ELSIF (F_BACnet_GetObjType(_ObjectId) <> BACnetObjectType_MultiStateOutput) THEN
	(* wrong mapping / invalid object ID *)
	IF _ObjectId = 0 THEN
		nErrorId := BACnet_ERR_WRONG_MAPPING;
	ELSE
		nErrorId := BACnet_ERR_INVALID_OBJECTID;
	END_IF
	bReady := FALSE;

ELSIF (_StatusFlags < 4) THEN
	(* wrong mapping *)
	nErrorId := BACnet_ERR_WRONG_MAPPING;
	bReady := FALSE;

ELSIF Device.bOperational THEN
	(* ready state *)
	bReady := TRUE;
	nErrorId := BACnet_ERR_NO_ERROR;

	(* write into priority array *)
	_PresentValue_Priority12 := F_BACnet_MultiStatePV(bEnablePV, bNullPV, nPV);

	(* present value *)
	nPresentValue := _PresentValue;

	(* build bit states *)
	_StatusFlagsBits := F_BACnet_StatusFlags(_StatusFlags);
	_AckedTransBits		:= F_BACnet_EventTransitionFlags(_AckedTransitions);

	(* copy states to output *)
	bOverridden := _StatusFlagsBits.overridden;
	bOutOfService := _StatusFlagsBits.out_of_service;
	bFault := _StatusFlagsBits.fault;
	bInAlarm := _StatusFlagsBits.in_alarm;
	bNoOutput := (_Reliability = TO_WORD(BACnetReliability_no_output));
	bOpenLoop := (_Reliability = TO_WORD(BACnetReliability_open_loop));
	bShortedLoop := (_Reliability = TO_WORD(BACnetReliability_shorted_loop));
	bOtherFault := (_Reliability = TO_WORD(BACnetReliability_unreliable_other));
	bAckedTrans_ToOffNormal := _AckedTransBits.to_offnormal;
	bAckedTrans_ToFault := _AckedTransBits.to_fault;
	bAckedTrans_ToNormal := _AckedTransBits.to_normal;
	tObjectID := _ObjectId;

	(* convert enumeration *)
	eEventState := TO_INT(_EventState);

	(* copy active priority *)
	nActivePrio := UDINT_TO_UINT(_ActivePriority);

	(* number of states *)
	nNbrOfStates := _NumberOfStates;

ELSE
	(* server device not ready, reset local ready also *)
	bReady := FALSE;
	nErrorId := BACnet_ERR_OPERATIONAL;
END_IF
(* set error flag *)
bError := (nErrorId <> BACnet_ERR_NO_ERROR);

END_FUNCTION_BLOCK

// POUs/BACnet Objects/Local (Server)/Extended Process Data/FB_BACnet_MultiStateValue_EX
FUNCTION_BLOCK FB_BACnet_MultiStateValue_EX
VAR_INPUT
	bEnablePV			: BOOL; (* enable present value with priority x in priority array, FALSE = priority x disable *)
	bNullPV				: BOOL; (* clear priority entry *)
	nPV					: UDINT; (* number for priority x, when input bEnablePV is TRUE *)
END_VAR
VAR_IN_OUT
	Device				: FB_BACnet_Device;
END_VAR
VAR_OUTPUT
	bReady				: BOOL;
	nPresentValue		: UDINT;
	bOverridden			: BOOL;
	bOutOfService		: BOOL;
	bFault				: BOOL;
	bInAlarm			: BOOL;
	bMultiStateFault	: BOOL;
	bOtherFault			: BOOL;
	eEventState			: E_BACNETEVENTSTATE;
	bAckedTrans_ToOffNormal : BOOL;
	bAckedTrans_ToFault		: BOOL;
	bAckedTrans_ToNormal	: BOOL;
	nActivePrio			: UINT;
	nNbrOfStates		: UDINT;
	tObjectID			: T_BACnet_ObjectIdentifier := 16#FFFFFFFF;
	bError				: BOOL;
	nErrorId			: UINT;
END_VAR
VAR
	_PresentValue AT%I*: UDINT; 			(* ~(BACnet_PresentValue 	:		: )
								   				(BACnet_ObjectType 		: MV	: )	*)
    _PresentValue_Priority12 AT%Q*: UDINT;	(* ~(BACnet_PresentValue_Priority12	:		: )	*)
	_ActivePriority AT%I*: UDINT; 			(* ~(BACnet_ActivePriority 	:		: )	*)
	_NumberOfStates AT%I*: UDINT;			(* ~(BACnet_NumberOfStates	:		: )	*)
	_ObjectId AT%I*: DWORD;					(* ~(BACnet_ObjectIdentifier:		: LINK) *)
	_StatusFlags AT%I*: WORD; 				(* ~(BACnet_StatusFlags 	:		: )	*)
	_EventState AT%I*: WORD;				(* ~(BACnet_EventState 		:		: )	*)
	_Reliability AT%I*: WORD;;				(* ~(BACnet_Reliability 	:		: )	*)
	_AckedTransitions AT%I*:WORD;			(* ~(BACnet_AckedTransitions:		: ) *)
	_AckedTransBits : ST_BACnet_EventTransitionBits;
	_StatusFlagsBits : ST_BACnet_StatusFlags;
	_nUpdateCount : UDINT := 0;
END_VAR

(* update server device *)
IF (Device._nUpdateCount = _nUpdateCount) THEN
	Device();
END_IF
(* remind current number of update counter *)
_nUpdateCount := Device._nUpdateCount;

IF Device.bFirstCycle THEN
	(* first call of the server device since reboot/reset *)
	bReady := FALSE;
	_PresentValue_Priority12 := 16#FFFFFFFF;

ELSIF (F_BACnet_GetObjType(_ObjectId) <> BACnetObjectType_MultiStateValue) THEN
	(* wrong mapping / invalid object ID *)
	IF _ObjectId = 0 THEN
		nErrorId := BACnet_ERR_WRONG_MAPPING;
	ELSE
		nErrorId := BACnet_ERR_INVALID_OBJECTID;
	END_IF
	bReady := FALSE;

ELSIF (_StatusFlags < 4) THEN
	(* wrong mapping *)
	nErrorId := BACnet_ERR_WRONG_MAPPING;
	bReady := FALSE;

ELSIF Device.bOperational THEN
	(* ready state *)
	bReady := TRUE;
	nErrorId := BACnet_ERR_NO_ERROR;

	(* write into priority array *)
	_PresentValue_Priority12 := F_BACnet_MultiStatePV(bEnablePV, bNullPV, nPV);

	(* present value *)
	nPresentValue := _PresentValue;

	(* build bit states *)
	_StatusFlagsBits := F_BACnet_StatusFlags(_StatusFlags);
	_AckedTransBits		:= F_BACnet_EventTransitionFlags(_AckedTransitions);

	(* copy states to output *)
	bOverridden := _StatusFlagsBits.overridden;
	bOutOfService := _StatusFlagsBits.out_of_service;
	bFault := _StatusFlagsBits.fault;
	bInAlarm := _StatusFlagsBits.in_alarm;
	bMultiStateFault := (_Reliability = TO_WORD(BACnetReliability_multi_state_fault));
	bOtherFault := (_Reliability = TO_WORD(BACnetReliability_unreliable_other));
	bAckedTrans_ToOffNormal := _AckedTransBits.to_offnormal;
	bAckedTrans_ToFault := _AckedTransBits.to_fault;
	bAckedTrans_ToNormal := _AckedTransBits.to_normal;
	tObjectID := _ObjectId;

	(* convert enumeration *)
	eEventState := TO_INT(_EventState);

	(* copy active priority *)
	nActivePrio := UDINT_TO_UINT(_ActivePriority);

	(* number of states *)
	nNbrOfStates := _NumberOfStates;

ELSE
	(* server device not ready, reset local ready also *)
	bReady := FALSE;
	nErrorId := BACnet_ERR_OPERATIONAL;
END_IF
(* set error flag *)
bError := (nErrorId <> BACnet_ERR_NO_ERROR);

END_FUNCTION_BLOCK

// POUs/BACnet Objects/Local (Server)/Extended Process Data/FB_BACnet_NotificationClass_EX
FUNCTION_BLOCK FB_BACnet_NotificationClass_EX
VAR_IN_OUT
	Device				: FB_BACnet_Device;
END_VAR
VAR_OUTPUT
	bReady				: BOOL;
	tObjectID			: T_BACnet_ObjectIdentifier := 16#FFFFFFFF;
	bError				: BOOL;
	nErrorId			: UINT;
END_VAR
VAR
	_ObjectId AT%I* : DWORD;					(* ~(BACnet_ObjectIdentifier:		: LINK)
													(BACnet_ObjectType		:	NC	: ) *)
	_nUpdateCount	: UDINT := 0;
END_VAR

(* update server device *)
IF (Device._nUpdateCount = _nUpdateCount) THEN
	Device();
END_IF
(* remind current number of update counter *)
_nUpdateCount := Device._nUpdateCount;

IF (F_BACnet_GetObjType(_ObjectId) <> BACnetObjectType_NotificationClass) THEN
	(* wrong mapping / invalid object ID *)
	IF _ObjectId = 0 THEN
		nErrorId := BACnet_ERR_WRONG_MAPPING;
	ELSE
		nErrorId := BACnet_ERR_INVALID_OBJECTID;
	END_IF
	bReady := FALSE;
	tObjectID := 16#FFFFFFFF;

ELSIF Device.bOperational THEN
	(* ready state *)
	bReady := TRUE;
	nErrorId := BACnet_ERR_NO_ERROR;
	tObjectID := _ObjectId;

ELSE
	(* server device not ready, reset local ready also *)
	bReady := FALSE;
	nErrorId := BACnet_ERR_OPERATIONAL;
END_IF
(* set error flag *)
bError := (nErrorId <> BACnet_ERR_NO_ERROR);

END_FUNCTION_BLOCK

// POUs/BACnet Objects/Local (Server)/Extended Process Data/FB_BACnet_Program_EX
FUNCTION_BLOCK FB_BACnet_Program_EX
VAR_INPUT
	bRelease			: BOOL;
	bCommonError		: BOOL;
	bWaitForSomething	: BOOL;
	stDoneFlags			: ST_BACnet_ProgramHandshakeRequests;
	stFailedFlags		: ST_BACnet_ProgramHandshakeRequests;
	bModeUnloadComplex	: BOOL := TRUE;
END_VAR
VAR_IN_OUT
	Device				: FB_BACnet_Device;
END_VAR
VAR_OUTPUT
	bReady				: BOOL;
	bOverridden			: BOOL;
	bOutOfService		: BOOL;
	bFault				: BOOL;
	bInAlarm			: BOOL;
	bProcessError		: BOOL;
	bCommFailure		: BOOL;
	bOtherFault			: BOOL;
	stRequestFlags		: ST_BACnet_ProgramHandshakeRequests;
	stActiveStateFlags	: ST_BACnet_ProgramHandshakeStates;
	tObjectID			: T_BACnet_ObjectIdentifier := 16#FFFFFFFF;
	bError				: BOOL;
	nErrorId			: UINT;
END_VAR
VAR
(* from BACnet to PLC *)
	_ObjectId AT%I* : DWORD;			(* ~(BACnet_ObjectIdentifier	:		: LINK) *)
	_ProgramChange AT%I*: WORD;			(* ~(BACnet_ProgramChange 		:		: )
											(BACnet_ObjectType 			: PROG	: ) *)
	_StatusFlags AT%I*: WORD;			(* ~(BACnet_StatusFlags 		:		: )	*)
	_Reliability AT%I*: WORD;;			(* ~(BACnet_Reliability 		:		: )	*)

(* from PLC to BACnet *)
	_ProgramState AT%Q*: WORD;			(* ~(BACnet_ProgramState 		:		: ) *)
	_ReasonForHalt AT%Q*: WORD;			(* ~(BACnet_ReasonForHalt 		:		: )	*)
	_SetProgramReadyState AT%Q*: BOOL;	(* ~(BACnet_SetProgramReadyState:		: )	*)

(* internal signals *)
	_StatusFlagsBits 	: ST_BACnet_StatusFlags;
	_bTriggerSetup		: BOOL;
	_ActiveChange		: E_BACNETPROGRAMREQUEST; (* ACTIVE PROGRAM CHANGE *)
	_bLockedForChange	: BOOL;
	_nUpdateCount		: UDINT := 0;
END_VAR

(* update server device *)
IF (Device._nUpdateCount = _nUpdateCount) THEN
	Device();
END_IF
(* remind current number of update counter *)
_nUpdateCount := Device._nUpdateCount;

(* check BitString format of StatusFlags --> if StatusFlags are less than 4, object isn't linked correctly *)
IF (F_BACnet_GetObjType(_ObjectId) <> BACnetObjectType_Program) THEN
	(* wrong mapping / invalid object ID *)
	IF _ObjectId = 0 THEN
		nErrorId := BACnet_ERR_WRONG_MAPPING;
	ELSE
		nErrorId := BACnet_ERR_INVALID_OBJECTID;
	END_IF
	bReady := FALSE;
	tObjectID := 16#FFFFFFFF;

ELSIF (_StatusFlags < 4) THEN
	(* wrong mapping *)
	nErrorId := BACnet_ERR_WRONG_MAPPING;
	bReady := FALSE;

ELSIF Device.bOperational THEN
	(* ready state *)
	bReady := TRUE;
	nErrorId := BACnet_ERR_NO_ERROR;

	(* decode status flags *)
	_StatusFlagsBits := F_BACnet_StatusFlags(_StatusFlags);

	(* copy states to output *)
	bOverridden := _StatusFlagsBits.overridden;
	bOutOfService := _StatusFlagsBits.out_of_service;
	bFault := _StatusFlagsBits.fault;
	bInAlarm := _StatusFlagsBits.in_alarm;
	bProcessError := (_Reliability = TO_WORD(BACnetReliability_process_error));
	bCommFailure := (_Reliability = TO_WORD(BACnetReliability_communication_failure));
	bOtherFault := (_Reliability = TO_WORD(BACnetReliability_unreliable_other));
	tObjectID := _ObjectId;

	(* execute change *)
	CASE _ActiveChange OF
		BACnetProgramRequest_ready:
			(* idle *);

		BACnetProgramRequest_load:
			_ProgramState	 := TO_WORD(BACnetProgramState_loading);
			_ActiveChange	:= BACnetProgramRequest_ready;

		BACnetProgramRequest_restart,
		BACnetProgramRequest_run:
			IF _bTriggerSetup THEN
				(* wait on setup finish *)
				IF stFailedFlags.bSetup OR bCommonError OR (NOT bRelease) THEN
					(* abort *)
					_ProgramState := TO_WORD(BACnetProgramState_halted);
					_ActiveChange := BACnetProgramRequest_ready;
					_ReasonForHalt  := TO_WORD(BACnetProgramError_progerror_internal);
				ELSIF stDoneFlags.bSetup THEN
					(* setup done, start "normal" running mode *)
					_bTriggerSetup := FALSE;
					_ActiveChange := BACnetProgramRequest_run;
				END_IF
			ELSE
				IF stFailedFlags.bRun OR bCommonError OR (NOT bRelease) THEN
					(* abort *)
					_ProgramState := TO_WORD(BACnetProgramState_halted);
					_ActiveChange := BACnetProgramRequest_ready;
					_ReasonForHalt  := TO_WORD(BACnetProgramError_progerror_internal);
				ELSIF stDoneFlags.bRun THEN
					(* switch to running state *)
					_ProgramState  := TO_WORD(BACnetProgramState_running);
					_ActiveChange := BACnetProgramRequest_ready;
				END_IF
			END_IF

		BACnetProgramRequest_halt:
			(* wait on halted *)
			IF stFailedFlags.bHalt OR bCommonError OR (NOT bRelease) THEN
				(* abort *)
				_ProgramState := TO_WORD(BACnetProgramState_halted);
				_ActiveChange := BACnetProgramRequest_ready;
				_ReasonForHalt  := TO_WORD(BACnetProgramError_progerror_internal);
			ELSIF stDoneFlags.bHalt THEN
				(* halted *)
				_ProgramState := TO_WORD(BACnetProgramState_halted);
				_ActiveChange := BACnetProgramRequest_ready;
				_ReasonForHalt  := TO_WORD(BACnetProgramError_program);
			END_IF

		BACnetProgramRequest_unload:
			_ProgramState	 := TO_WORD(BACnetProgramState_unloading);
			_ActiveChange	:= BACnetProgramRequest_ready;

	END_CASE

	(* start change request and handle error states *)
	IF (_ActiveChange = BACnetProgramRequest_ready) THEN

		CASE TO_DINT(_ProgramState) OF
			BACnetProgramState_idle:
				IF bCommonError THEN
					(* abort *)
					_ProgramState := TO_WORD(BACnetProgramState_halted);
					_ReasonForHalt  := TO_WORD(BACnetProgramError_progerror_internal);
				ELSIF (NOT bRelease) THEN
					(* abort *)
					_ProgramState := TO_WORD(BACnetProgramState_halted);
					_ReasonForHalt  := TO_WORD(BACnetProgramError_other);
				ELSIF (NOT _bLockedForChange) THEN
					_ReasonForHalt  := TO_WORD(BACnetProgramError_program_normal);
					CASE to_dint(_ProgramChange) OF
						BACnetProgramRequest_unload,
						BACnetProgramRequest_halt:
							(* acknowledge without execution *)
							_SetProgramReadyState	:= TRUE;
						BACnetProgramRequest_restart,
						BACnetProgramRequest_run,
						BACnetProgramRequest_load:
							(* execute request *)
							_ActiveChange := BACnetProgramRequest_load;
							_bTriggerSetup := TRUE;
					END_CASE
				END_IF

			BACnetProgramState_loading:
				IF bCommonError THEN
					(* abort *)
					_ProgramState := TO_WORD(BACnetProgramState_halted);
					_ReasonForHalt  := TO_WORD(BACnetProgramError_progerror_internal);
				ELSIF (NOT bRelease) THEN
					(* abort *)
					_ProgramState := TO_WORD(BACnetProgramState_halted);
					_ReasonForHalt  := TO_WORD(BACnetProgramError_other);
				ELSIF stFailedFlags.bLoad THEN
					(* abort *)
					_ProgramState := TO_WORD(BACnetProgramState_halted);
					_ReasonForHalt  := TO_WORD(BACnetProgramError_load_failed);
				ELSIF stDoneFlags.bLoad THEN
					(* DONE *)
					_bTriggerSetup := TRUE;
					_ActiveChange := BACnetProgramRequest_run;
				ELSIF (NOT _bLockedForChange) THEN
					_ReasonForHalt  := TO_WORD(BACnetProgramError_program_normal);
					CASE TO_DINT(_ProgramChange) OF
						BACnetProgramRequest_load,
						BACnetProgramRequest_run,
						BACnetProgramRequest_halt,
						BACnetProgramRequest_restart:
							(* acknowledge without execution *)
							_SetProgramReadyState	:= TRUE;
						BACnetProgramRequest_unload:
							(* execute request *)
							_ActiveChange := to_int(_ProgramChange);
					END_CASE
				END_IF

			BACnetProgramState_running:
				IF bCommonError THEN
					(* abort *)
					_ProgramState := TO_WORD(BACnetProgramState_halted);
					_ReasonForHalt  := TO_WORD(BACnetProgramError_progerror_internal);
				ELSIF (NOT bRelease) THEN
					(* abort *)
					_ProgramState := TO_WORD(BACnetProgramState_halted);
					_ReasonForHalt  := TO_WORD(BACnetProgramError_other);
				ELSIF bWaitForSomething THEN
					(* wait on something *)
					_ProgramState  := TO_WORD(BACnetProgramState_waiting);
				ELSIF (NOT _bLockedForChange) THEN
					_ReasonForHalt  := TO_WORD(BACnetProgramError_program_normal);
					CASE to_dint(_ProgramChange) OF
						BACnetProgramRequest_run:
							(* is already running *)
							_SetProgramReadyState	:= TRUE;
						BACnetProgramRequest_unload,
						BACnetProgramRequest_halt:
							(* execute request *)
							_ActiveChange := to_int(_ProgramChange);
						BACnetProgramRequest_restart,
						BACnetProgramRequest_load:
							(* retrigger setup *)
							_ActiveChange := BACnetProgramRequest_restart;
							_bTriggerSetup := TRUE;
					END_CASE
				END_IF

			BACnetProgramState_waiting:
				IF bCommonError THEN
					(* abort *)
					_ProgramState := TO_WORD(BACnetProgramState_halted);
					_ReasonForHalt  := TO_WORD(BACnetProgramError_progerror_internal);
				ELSIF (NOT bRelease) THEN
					(* abort *)
					_ProgramState := TO_WORD(BACnetProgramState_halted);
					_ReasonForHalt  := TO_WORD(BACnetProgramError_other);
				ELSIF (NOT bWaitForSomething) THEN
					(* got it *)
					_ProgramState  := TO_WORD(BACnetProgramState_running);
				ELSIF (NOT _bLockedForChange) THEN
					_ReasonForHalt  := TO_WORD(BACnetProgramError_program_normal);
					CASE to_dint(_ProgramChange) OF
						BACnetProgramRequest_run:
							(* is already running *)
							_SetProgramReadyState	:= TRUE;
						BACnetProgramRequest_unload,
						BACnetProgramRequest_halt:
							(* execute request *)
							_ActiveChange := to_int(_ProgramChange);
					END_CASE
				END_IF

			BACnetProgramState_halted:
				IF (NOT bCommonError) AND bRelease AND (NOT _bLockedForChange) THEN
					CASE to_dint(_ProgramChange) OF
						BACnetProgramRequest_halt:
							(* acknowledge without execution *)
							_SetProgramReadyState	:= TRUE;
						BACnetProgramRequest_unload:
							(* execute request *)
							_ActiveChange := to_int(_ProgramChange);
						BACnetProgramRequest_restart,
						BACnetProgramRequest_load:
							(* retrigger setup *)
							_ActiveChange := BACnetProgramRequest_restart;
							_bTriggerSetup := TRUE;
						BACnetProgramRequest_run:
							(* start, but don't trigger setup *)
							_ActiveChange := to_int(_ProgramChange);
							_bTriggerSetup := FALSE;
					END_CASE
				END_IF

			BACnetProgramState_unloading:
				IF bModeUnloadComplex THEN
					_ReasonForHalt  := TO_WORD(BACnetProgramError_program_normal);
					IF bCommonError THEN
						(* abort *)
						_ProgramState := TO_WORD(BACnetProgramState_halted);
						_ActiveChange := BACnetProgramRequest_ready;
						_ReasonForHalt  := TO_WORD(BACnetProgramError_progerror_internal);
					ELSIF (NOT bRelease) THEN
						(* abort *)
						_ProgramState := TO_WORD(BACnetProgramState_halted);
						_ActiveChange := BACnetProgramRequest_ready;
						_ReasonForHalt  := TO_WORD(BACnetProgramError_other);
					ELSIF stFailedFlags.bUnload THEN
						(* abort *)
						_ProgramState := TO_WORD(BACnetProgramState_halted);
						_ActiveChange := BACnetProgramRequest_ready;
						_ReasonForHalt  := TO_WORD(BACnetProgramError_other);
					ELSIF stDoneFlags.bUnload THEN
						(* DONE *)
						_ActiveChange := BACnetProgramRequest_ready;
						_ProgramState  := TO_WORD(BACnetProgramState_idle);
					ELSIF (NOT _bLockedForChange) THEN
						CASE to_dint(_ProgramChange) OF
							BACnetProgramRequest_load,
							BACnetProgramRequest_run,
							BACnetProgramRequest_halt,
							BACnetProgramRequest_restart,
							BACnetProgramRequest_unload:
								(* acknowledge without execution *)
								_SetProgramReadyState	:= TRUE;
						END_CASE
					END_IF
				END_IF

		END_CASE
	END_IF

	(* check state of "change" request *)
	IF (_ActiveChange <> BACnetProgramRequest_ready) THEN
		(* request is active, lock execution *)
		_bLockedForChange		:= TRUE;
	ELSIF _bLockedForChange AND (NOT _SetProgramReadyState) THEN
		(* change finished, tell the stack done *)
		_SetProgramReadyState	:= TRUE;
		_bTriggerSetup			:= FALSE;
	ELSIF (_ProgramChange = TO_WORD(BACnetProgramRequest_ready)) THEN
		(* wait on new requests *)
		_SetProgramReadyState	:= FALSE;
		_bLockedForChange		:= FALSE;
		_bTriggerSetup			:= FALSE;
	ELSE
		(* new request *)
		_bTriggerSetup			:= FALSE;
	END_IF

	(* external requests *)
	stRequestFlags.bLoad			:= _ProgramState = to_word(TO_WORD(BACnetProgramState_loading)) AND (NOT _bLockedForChange);
	stRequestFlags.bSetup			:=	(		(_ActiveChange = BACnetProgramRequest_run)
										OR	(_ActiveChange = BACnetProgramRequest_restart)
									)
								AND	_bTriggerSetup;
	stRequestFlags.bRun			:= (_ActiveChange = BACnetProgramRequest_run) AND (NOT _bTriggerSetup);
	stRequestFlags.bHalt			:= _ActiveChange = BACnetProgramRequest_halt;
	stRequestFlags.bUnload		:=	(_ActiveChange = BACnetProgramRequest_unload)
								OR	(		_ProgramState = to_word(TO_WORD(BACnetProgramState_unloading))
										AND	(NOT _bLockedForChange)
									);

	(* active status flags *)
	stActiveStateFlags.bIdle		:= _ProgramState = TO_WORD(BACnetProgramState_idle);
	stActiveStateFlags.bLoading		:= _ProgramState = TO_WORD(BACnetProgramState_loading);
	stActiveStateFlags.bRunning		:= _ProgramState = TO_WORD(BACnetProgramState_running);
	stActiveStateFlags.bWaiting		:= _ProgramState = TO_WORD(BACnetProgramState_waiting);
	stActiveStateFlags.bHalted		:= _ProgramState = TO_WORD(BACnetProgramState_halted);
	stActiveStateFlags.bUnloading	:= _ProgramState = TO_WORD(BACnetProgramState_unloading);
ELSE
	(* server device not ready, reset local ready also *)
	bReady := FALSE;
	nErrorId := BACnet_ERR_OPERATIONAL;
END_IF
(* set error flag *)
bError := (nErrorId <> BACnet_ERR_NO_ERROR);

END_FUNCTION_BLOCK

